(* POU FB_BACnet_MultiStateOutput_EX, ST *)
FUNCTION_BLOCK FB_BACnet_MultiStateOutput_EX
VAR_INPUT
	bEnablePV			: BOOL; (* enable present value with priority x in priority array, FALSE = priority x disable *)
	bNullPV				: BOOL; (* clear priority entry *)
	nPV					: UDINT; (* number for priority x, when input bEnablePV is TRUE *)
END_VAR
VAR_IN_OUT
	Device				: FB_BACnet_Device;
END_VAR
VAR_OUTPUT
	bReady				: BOOL;
	nPresentValue		: UDINT;
	bOverridden			: BOOL;
	bOutOfService		: BOOL;
	bFault				: BOOL;
	bInAlarm			: BOOL;
	bNoOutput			: BOOL;
	bOpenLoop			: BOOL;
	bShortedLoop		: BOOL;
	bOtherFault			: BOOL;
	eEventState			: E_BACNETEVENTSTATE;
	bAckedTrans_ToOffNormal : BOOL;
	bAckedTrans_ToFault		: BOOL;
	bAckedTrans_ToNormal	: BOOL;
	nActivePrio			: UINT;
	nNbrOfStates		: UDINT;
	tObjectID			: T_BACnet_ObjectIdentifier := 16#FFFFFFFF;
	bError				: BOOL;
	nErrorId			: UINT;
END_VAR
VAR
	_PresentValue AT%I*: UDINT; 			(* ~(BACnet_PresentValue 		:		: )
								   				(BACnet_ObjectType			: MO	: )	*)
    _PresentValue_Priority12 AT%Q*: UDINT;	(* ~(BACnet_PresentValue_Priority12		:		: )	*)
	_ActivePriority AT%I*: UDINT; 			(* ~(BACnet_ActivePriority 		:		: )	*)
	_NumberOfStates AT%I*: UDINT;			(* ~(BACnet_NumberOfStates		:		: )	*)
	_ObjectId AT%I*: DWORD;					(* ~(BACnet_ObjectIdentifier	:		: LINK) *)
	_StatusFlags AT%I*: WORD; 				(* ~(BACnet_StatusFlags			:		: )	*)
	_EventState AT%I*: WORD;				(* ~(BACnet_EventState			:		: )	*)
	_Reliability AT%I*: WORD; 				(* ~(BACnet_Reliability			:		: )	*)
	_AckedTransitions AT%I*:WORD;			(* ~(BACnet_AckedTransitions	:		: ) *)
	_AckedTransBits : ST_BACnet_EventTransitionBits;
	_nUpdateCount : UDINT := 0;
	_StatusFlagsBits : ST_BACnet_StatusFlags;
END_VAR
(* update server device *)
IF (Device._nUpdateCount = _nUpdateCount) THEN
	Device();
END_IF
(* remind current number of update counter *)
_nUpdateCount := Device._nUpdateCount;

IF Device.bFirstCycle THEN
	(* first call of the server device since reboot/reset *)
	bReady := FALSE;
	_PresentValue_Priority12 := 16#FFFFFFFF;

ELSIF (F_BACnet_GetObjType(_ObjectId) <> BACnetObjectType_MultiStateOutput) THEN
	(* wrong mapping / invalid object ID *)
	IF _ObjectId = 0 THEN
		nErrorId := BACnet_ERR_WRONG_MAPPING;
	ELSE
		nErrorId := BACnet_ERR_INVALID_OBJECTID;
	END_IF
	bReady := FALSE;

ELSIF (_StatusFlags < 4) THEN
	(* wrong mapping *)
	nErrorId := BACnet_ERR_WRONG_MAPPING;
	bReady := FALSE;

ELSIF Device.bOperational THEN
	(* ready state *)
	bReady := TRUE;
	nErrorId := BACnet_ERR_NO_ERROR;

	(* write into priority array *)
	_PresentValue_Priority12 := F_BACnet_MultiStatePV(bEnablePV, bNullPV, nPV);

	(* present value *)
	nPresentValue := _PresentValue;

	(* build bit states *)
	_StatusFlagsBits := F_BACnet_StatusFlags(_StatusFlags);
	_AckedTransBits		:= F_BACnet_EventTransitionFlags(_AckedTransitions);

	(* copy states to output *)
	bOverridden := _StatusFlagsBits.overridden;
	bOutOfService := _StatusFlagsBits.out_of_service;
	bFault := _StatusFlagsBits.fault;
	bInAlarm := _StatusFlagsBits.in_alarm;
	bNoOutput := (_Reliability = BACnetReliability_no_output);
	bOpenLoop := (_Reliability = BACnetReliability_open_loop);
	bShortedLoop := (_Reliability = BACnetReliability_shorted_loop);
	bOtherFault := (_Reliability = BACnetReliability_unreliable_other);
	bAckedTrans_ToOffNormal := _AckedTransBits.to_offnormal;
	bAckedTrans_ToFault := _AckedTransBits.to_fault;
	bAckedTrans_ToNormal := _AckedTransBits.to_normal;
	tObjectID := _ObjectId;

	(* convert enumeration *)
	eEventState := _EventState;

	(* copy active priority *)
	nActivePrio := UDINT_TO_UINT(_ActivePriority);

	(* number of states *)
	nNbrOfStates := _NumberOfStates;

ELSE
	(* server device not ready, reset local ready also *)
	bReady := FALSE;
	nErrorId := BACnet_ERR_OPERATIONAL;
END_IF
(* set error flag *)
bError := (nErrorId <> BACnet_ERR_NO_ERROR);
END_FUNCTION_BLOCK

(* POU FB_BACnet_MultiStateOutput_RAW, ST *)
FUNCTION_BLOCK FB_BACnet_MultiStateOutput_RAW
VAR_INPUT
	bEnablePV			: BOOL; (* enable present value with priority x in priority array, FALSE = priority x disable *)
	bNullPV				: BOOL; (* clear priority entry *)
	nPV					: UDINT; (* number for priority x, when input bEnablePV is TRUE *)
	nFeedback			AT%Q*: DWORD; (* ~(BACnet_FeedbackValue : : ) *)
	bNoOutput			: BOOL;
	bOpenLoop			: BOOL;
	bShortedLoop		: BOOL;
	bCommFailure		: BOOL;
	bOtherFault			: BOOL;
END_VAR
VAR_IN_OUT
	Device				: FB_BACnet_Device;
END_VAR
VAR_OUTPUT
	bReady				: BOOL;
	nPresentValue		: UDINT;
	bOverridden			: BOOL;
	bOutOfService		: BOOL;
	bFault				: BOOL;
	bInAlarm			: BOOL;
	bAckedTrans_ToOffNormal : BOOL;
	bAckedTrans_ToFault		: BOOL;
	bAckedTrans_ToNormal	: BOOL;
	nNbrOfStates		: UDINT;
	bError				: BOOL;
	nErrorId			: UINT;
	nRawOut				AT%I*: DWORD;		(* ~(BACnet_PresentValue		:		: ) *)
END_VAR
VAR
    _PresentValue_Priority12 AT%Q*: UDINT;	(* ~(BACnet_PresentValue_Priority12:	: )
								   				(BACnet_ObjectType			: MO	: )	*)
	_Reliability AT%Q*: WORD := BACnetReliability_no_fault_detected;(* ~(BACnet_Reliability 	:		: )	*)
	_NumberOfStates AT%I*: UDINT;			(* ~(BACnet_NumberOfStates		:		: )	*)
	_ObjectId AT%I*: DWORD;					(* ~(BACnet_ObjectIdentifier	:		: LINK) *)
	_StatusFlags AT%I*: WORD; 				(* ~(BACnet_StatusFlags			:		: )	*)
	_AckedTransitions AT%I*:WORD;			(* ~(BACnet_AckedTransitions	:		: ) *)
	_AckedTransBits : ST_BACnet_EventTransitionBits;
	_nUpdateCount : UDINT := 0;
	_StatusFlagsBits : ST_BACnet_StatusFlags;
END_VAR
(* update server device *)
IF (Device._nUpdateCount = _nUpdateCount) THEN
	Device();
END_IF
(* remind current number of update counter *)
_nUpdateCount := Device._nUpdateCount;

(* handle raw error *)
IF bNoOutput THEN
	_Reliability := BACnetReliability_no_output;
ELSIF bOpenLoop THEN
	_Reliability := BACnetReliability_open_loop;
ELSIF bShortedLoop THEN
	_Reliability := BACnetReliability_shorted_loop;
ELSIF bCommFailure THEN
	_Reliability := BACnetReliability_communication_failure;
ELSIF bOtherFault THEN
	_Reliability := BACnetReliability_unreliable_other;
ELSE
	_Reliability := BACnetReliability_no_fault_detected;
END_IF

(* check object type *)
IF Device.bFirstCycle THEN
	(* first call of the server device since reboot/reset *)
	bReady := FALSE;
	_PresentValue_Priority12 := 16#FFFFFFFF;

ELSIF (F_BACnet_GetObjType(_ObjectId) <> BACnetObjectType_MultiStateOutput) THEN
	(* wrong mapping / invalid object ID *)
	IF _ObjectId = 0 THEN
		nErrorId := BACnet_ERR_WRONG_MAPPING;
	ELSE
		nErrorId := BACnet_ERR_INVALID_OBJECTID;
	END_IF
	bReady := FALSE;

ELSIF (_StatusFlags < 4) THEN
	(* wrong mapping *)
	nErrorId := BACnet_ERR_WRONG_MAPPING;
	bReady := FALSE;

ELSIF Device.bOperational THEN
	(* ready state *)
	bReady := TRUE;
	nErrorId := BACnet_ERR_NO_ERROR;

	(* write into priority array *)
	_PresentValue_Priority12 := F_BACnet_MultiStatePV(bEnablePV, bNullPV, nPV);

	(* present value *)
	nPresentValue := nRawOut;

	(* build bit states *)
	_StatusFlagsBits := F_BACnet_StatusFlags(_StatusFlags);
	_AckedTransBits		:= F_BACnet_EventTransitionFlags(_AckedTransitions);

	(* copy states to output *)
	bOverridden := _StatusFlagsBits.overridden;
	bOutOfService := _StatusFlagsBits.out_of_service;
	bFault := _StatusFlagsBits.fault;
	bInAlarm := _StatusFlagsBits.in_alarm;
	bAckedTrans_ToOffNormal := _AckedTransBits.to_offnormal;
	bAckedTrans_ToFault := _AckedTransBits.to_fault;
	bAckedTrans_ToNormal := _AckedTransBits.to_normal;

	(* number of states *)
	nNbrOfStates := _NumberOfStates;

ELSE
	(* server device not ready, reset local ready also *)
	bReady := FALSE;
	nErrorId := BACnet_ERR_OPERATIONAL;
END_IF
(* set error flag *)
bError := (nErrorId <> BACnet_ERR_NO_ERROR);
END_FUNCTION_BLOCK

(* POU FB_BACnet_MultiStateValue, ST *)
FUNCTION_BLOCK FB_BACnet_MultiStateValue
VAR_INPUT
	bEnablePV		: BOOL; (* enable present value with priority x in priority array, FALSE = priority x disable *)
	bNullPV			: BOOL; (* clear priority entry *)
	nPV				: UDINT; (* number for priority x, when input bEnablePV is TRUE *)
END_VAR
VAR_IN_OUT
	Device	: FB_BACnet_Device;
END_VAR
VAR_OUTPUT
	bReady			: BOOL;
	nPresentValue	: UDINT;
	bOverridden		: BOOL;
	bOutOfService	: BOOL;
	bFault			: BOOL;
	bInAlarm		: BOOL;
	nNbrOfStates	: UDINT;
	bError			: BOOL;
	nErrorId		: UINT;
END_VAR
VAR
	_PresentValue AT%I*: UDINT; 			(* ~(BACnet_PresentValue 		:		: )
								   				(BACnet_ObjectType 			: MV	: )	*)
	_NumberOfStates AT%I*: UDINT;			(* ~(BACnet_NumberOfStates		:		: )	*)
	_StatusFlags AT%I*: WORD; 				(* ~(BACnet_StatusFlags 		:		: )	*)
    _PresentValue_Priority12 AT%Q*: UDINT;	(* ~(BACnet_PresentValue_Priority12:	: )	*)
	_nUpdateCount : UDINT := 0;
	_StatusFlagsBits : ST_BACnet_StatusFlags;
END_VAR
(* update server device *)
IF (Device._nUpdateCount = _nUpdateCount) THEN
	Device();
END_IF
(* remind current number of update counter *)
_nUpdateCount := Device._nUpdateCount;

IF Device.bFirstCycle THEN
	(* first call of the server device since reboot/reset *)
	bReady := FALSE;
	_PresentValue_Priority12 := 16#FFFFFFFF;

ELSIF (_StatusFlags < 4) THEN
	(* wrong mapping *)
	nErrorId := BACnet_ERR_WRONG_MAPPING;
	bReady := FALSE;

ELSIF Device.bOperational THEN
	(* ready state *)
	bReady := TRUE;
	nErrorId := BACnet_ERR_NO_ERROR;

	(* write into priority array *)
	_PresentValue_Priority12 := F_BACnet_MultiStatePV(bEnablePV, bNullPV, nPV);

	(* present value *)
	nPresentValue := _PresentValue;

	(* build bit states *)
	_StatusFlagsBits := F_BACnet_StatusFlags(_StatusFlags);

	(* copy states to output *)
	bOverridden := _StatusFlagsBits.overridden;
	bOutOfService := _StatusFlagsBits.out_of_service;
	bFault := _StatusFlagsBits.fault;
	bInAlarm := _StatusFlagsBits.in_alarm;

	(* number of states *)
	nNbrOfStates := _NumberOfStates;

ELSE
	(* server device not ready, reset local ready also *)
	bReady := FALSE;
	nErrorId := BACnet_ERR_OPERATIONAL;
END_IF
(* set error flag *)
bError := (nErrorId <> BACnet_ERR_NO_ERROR);
END_FUNCTION_BLOCK

(* POU FB_BACnet_MultiStateValue_ADS, ST *)
FUNCTION_BLOCK FB_BACnet_MultiStateValue_ADS
VAR_INPUT
	bEnablePV			: BOOL; (* enable PV write commands *)
	bNullPV				: BOOL; (* clear priority entry *)
	nPV					: UDINT; (* number for priority x, when input bEnablePV is TRUE and bNullPV is FALSE *)
	bManual				: BOOL; (* FALSE --> TRUE: write present_value immediately, FALSE: only write present_value on-change, TRUE: write present_value on-change and when device turns operational *)
	ePriority			: E_BACNETPRIORITY := BACNETPRIORITY_12;
END_VAR
VAR_IN_OUT
	Device				: FB_BACnet_Device;
END_VAR
VAR_OUTPUT
	bReady				: BOOL;
	bPvDone				: BOOL; (* present_value written over ADS *)
	nPresentValue		: UDINT;
	bOverridden			: BOOL;
	bOutOfService		: BOOL;
	bFault				: BOOL;
	bInAlarm			: BOOL;
	nNbrOfStates		: UDINT;
	tObjectID			: T_BACnet_ObjectIdentifier := 16#FFFFFFFF;
	bError				: BOOL;
	nErrorId			: UINT;
	nAdsErrorId			: UDINT;
END_VAR
VAR
	_StatusFlags AT%I*: WORD; 				(* ~(BACnet_StatusFlags 	:		: )	*)
	_PresentValue AT%I*: UDINT; 			(* ~(BACnet_PresentValue 	:		: )
								   				(BACnet_ObjectType 		: MV	: )	*)
	_NumberOfStates AT%I*: UDINT;			(* ~(BACnet_NumberOfStates	:		: )	*)
	_ObjectId AT%I*: DWORD;					(* ~(BACnet_ObjectIdentifier:		: LINK) *)
	_StatusFlagsBits : ST_BACnet_StatusFlags;
    _PresentValue_Ads : UDINT;
	_nUpdateCount : UDINT := 0;
	_WriteProp : FB_BACnet_WriteProp;
	_rtrigManual : R_TRIG;
	_bNullPvOld : BOOL;
	_nObjType : E_BACNETOBJECTTYPE;
END_VAR
(* update server device *)
IF (Device._nUpdateCount = _nUpdateCount) THEN
	Device();
END_IF
(* remind current number of update counter *)
_nUpdateCount := Device._nUpdateCount;

(* trigger on manual flag *)
_rtrigManual(CLK:= bManual, Q=> );

(* decode object type *)
_nObjType := F_BACnet_GetObjType(_ObjectId);

IF Device.bFirstCycle THEN
	(* first call of the server device since reboot/reset *)
	bReady := FALSE;
	bPvDone := FALSE;

ELSIF _nObjType <> BACnetObjectType_MultiStateValue THEN
	(* wrong mapped object type *)
	nErrorId := BACnet_ERR_INVALID_OBJECTTYPE;
	bReady := FALSE;
	bPvDone := FALSE;

ELSIF (_StatusFlags < 4) THEN
	(* wrong mapping *)
	nErrorId := BACnet_ERR_WRONG_MAPPING;
	bReady := FALSE;
	bPvDone := FALSE;

ELSIF Device.bOperational THEN

	IF Device.stAdsConn.bValid THEN
		(* write present_value on manual trigger, on-change and on operational recover *)
		IF		bEnablePV
			AND	(		_rtrigManual.Q
					OR	(nPV <> _PresentValue_Ads)
					OR	((NOT bReady) AND bManual)
					OR	(bNullPV <> _bNullPvOld)
				)
		THEN
			_WriteProp.bExecute := TRUE;
			bPvDone := FALSE;
			(* write depending on enable state *)
			IF bNullPV THEN
				_PresentValue_Ads := 0;
			ELSE
				_PresentValue_Ads := nPV;
			END_IF
			_bNullPvOld := bNullPV;
		END_IF

		(* ready state *)
		IF (nAdsErrorId = 0) THEN
			bReady := TRUE;
			nErrorId := BACnet_ERR_NO_ERROR;
		END_IF

	ELSE
		(* invalid ADS connection *)
		bReady := FALSE;
		nErrorId := BACnet_ERR_INVALID_ADS_CONN;
		bPvDone := FALSE;
	END_IF

	(* present value *)
	nPresentValue := _PresentValue;

	(* build bit states *)
	_StatusFlagsBits := F_BACnet_StatusFlags(_StatusFlags);

	(* copy states to output *)
	bOverridden := _StatusFlagsBits.overridden;
	bOutOfService := _StatusFlagsBits.out_of_service;
	bFault := _StatusFlagsBits.fault;
	bInAlarm := _StatusFlagsBits.in_alarm;
	tObjectID := _ObjectId;

	(* number of states *)
	nNbrOfStates := _NumberOfStates;

ELSE
	(* server device not ready, reset local ready also *)
	bReady := FALSE;
	nErrorId := BACnet_ERR_OPERATIONAL;
	bPvDone := FALSE;
END_IF

(* call write property command *)
_WriteProp(
	BACnetDevicePort	:= Device.stAdsConn.nAmsPort,
	bExecute			:= ,
	sNetId				:= Device.stAdsConn.sAmsNetId,
	ObjectType			:= _nObjType,
	PropertyID			:= BACnetPropertyIdentifier_PresentValue,
	Priority			:= ePriority,
	DataType			:= BACnetDataType_UnsignedInteger,
	ObjectInstance		:= F_BACnet_GetObjInstance(_ObjectId),
	ptrValue			:= ADR(_PresentValue_Ads),
	nLenValue			:= SIZEOF(_PresentValue_Ads),
	bDone				=> ,
	bBusy				=> ,
	bError				=> ,
	nErrID				=> );

(* set done flag *)
IF _WriteProp.bExecute AND (NOT _WriteProp.bBusy) THEN
	(* check if command was finished with error *)
	IF _WriteProp.bError THEN
		bPvDone		:= FALSE;
		bReady		:= FALSE;
		nErrorId	:= BACnet_ERR_ADS_Write;
	ELSE
		(* successful written *)
		bPvDone		:= TRUE;
	END_IF
	nAdsErrorId := _WriteProp.nErrID;
	(* reset execution bit *)
	_WriteProp(bExecute := FALSE);
END_IF

(* set error flag *)
bError := (nErrorId <> BACnet_ERR_NO_ERROR) OR (nAdsErrorId <> 0);
END_FUNCTION_BLOCK

(* POU FB_BACnet_MultiStateValue_EX, ST *)
FUNCTION_BLOCK FB_BACnet_MultiStateValue_EX
VAR_INPUT
	bEnablePV			: BOOL; (* enable present value with priority x in priority array, FALSE = priority x disable *)
	bNullPV				: BOOL; (* clear priority entry *)
	nPV					: UDINT; (* number for priority x, when input bEnablePV is TRUE *)
END_VAR
VAR_IN_OUT
	Device				: FB_BACnet_Device;
END_VAR
VAR_OUTPUT
	bReady				: BOOL;
	nPresentValue		: UDINT;
	bOverridden			: BOOL;
	bOutOfService		: BOOL;
	bFault				: BOOL;
	bInAlarm			: BOOL;
	bMultiStateFault	: BOOL;
	bOtherFault			: BOOL;
	eEventState			: E_BACNETEVENTSTATE;
	bAckedTrans_ToOffNormal : BOOL;
	bAckedTrans_ToFault		: BOOL;
	bAckedTrans_ToNormal	: BOOL;
	nActivePrio			: UINT;
	nNbrOfStates		: UDINT;
	tObjectID			: T_BACnet_ObjectIdentifier := 16#FFFFFFFF;
	bError				: BOOL;
	nErrorId			: UINT;
END_VAR
VAR
	_PresentValue AT%I*: UDINT; 			(* ~(BACnet_PresentValue 	:		: )
								   				(BACnet_ObjectType 		: MV	: )	*)
    _PresentValue_Priority12 AT%Q*: UDINT;	(* ~(BACnet_PresentValue_Priority12	:		: )	*)
	_ActivePriority AT%I*: UDINT; 			(* ~(BACnet_ActivePriority 	:		: )	*)
	_NumberOfStates AT%I*: UDINT;			(* ~(BACnet_NumberOfStates	:		: )	*)
	_ObjectId AT%I*: DWORD;					(* ~(BACnet_ObjectIdentifier:		: LINK) *)
	_StatusFlags AT%I*: WORD; 				(* ~(BACnet_StatusFlags 	:		: )	*)
	_EventState AT%I*: WORD;				(* ~(BACnet_EventState 		:		: )	*)
	_Reliability AT%I*: WORD;				(* ~(BACnet_Reliability 	:		: )	*)
	_AckedTransitions AT%I*:WORD;			(* ~(BACnet_AckedTransitions:		: ) *)
	_AckedTransBits : ST_BACnet_EventTransitionBits;
	_StatusFlagsBits : ST_BACnet_StatusFlags;
	_nUpdateCount : UDINT := 0;
END_VAR
(* update server device *)
IF (Device._nUpdateCount = _nUpdateCount) THEN
	Device();
END_IF
(* remind current number of update counter *)
_nUpdateCount := Device._nUpdateCount;

IF Device.bFirstCycle THEN
	(* first call of the server device since reboot/reset *)
	bReady := FALSE;
	_PresentValue_Priority12 := 16#FFFFFFFF;

ELSIF (F_BACnet_GetObjType(_ObjectId) <> BACnetObjectType_MultiStateValue) THEN
	(* wrong mapping / invalid object ID *)
	IF _ObjectId = 0 THEN
		nErrorId := BACnet_ERR_WRONG_MAPPING;
	ELSE
		nErrorId := BACnet_ERR_INVALID_OBJECTID;
	END_IF
	bReady := FALSE;

ELSIF (_StatusFlags < 4) THEN
	(* wrong mapping *)
	nErrorId := BACnet_ERR_WRONG_MAPPING;
	bReady := FALSE;

ELSIF Device.bOperational THEN
	(* ready state *)
	bReady := TRUE;
	nErrorId := BACnet_ERR_NO_ERROR;

	(* write into priority array *)
	_PresentValue_Priority12 := F_BACnet_MultiStatePV(bEnablePV, bNullPV, nPV);

	(* present value *)
	nPresentValue := _PresentValue;

	(* build bit states *)
	_StatusFlagsBits := F_BACnet_StatusFlags(_StatusFlags);
	_AckedTransBits		:= F_BACnet_EventTransitionFlags(_AckedTransitions);

	(* copy states to output *)
	bOverridden := _StatusFlagsBits.overridden;
	bOutOfService := _StatusFlagsBits.out_of_service;
	bFault := _StatusFlagsBits.fault;
	bInAlarm := _StatusFlagsBits.in_alarm;
	bMultiStateFault := (_Reliability = BACnetReliability_multi_state_fault);
	bOtherFault := (_Reliability = BACnetReliability_unreliable_other);
	bAckedTrans_ToOffNormal := _AckedTransBits.to_offnormal;
	bAckedTrans_ToFault := _AckedTransBits.to_fault;
	bAckedTrans_ToNormal := _AckedTransBits.to_normal;
	tObjectID := _ObjectId;

	(* convert enumeration *)
	eEventState := _EventState;

	(* copy active priority *)
	nActivePrio := UDINT_TO_UINT(_ActivePriority);

	(* number of states *)
	nNbrOfStates := _NumberOfStates;

ELSE
	(* server device not ready, reset local ready also *)
	bReady := FALSE;
	nErrorId := BACnet_ERR_OPERATIONAL;
END_IF
(* set error flag *)
bError := (nErrorId <> BACnet_ERR_NO_ERROR);
END_FUNCTION_BLOCK

(* POU FB_BACnet_NotificationClass, ST *)
FUNCTION_BLOCK FB_BACnet_NotificationClass
VAR_IN_OUT
	Device	: FB_BACnet_Device;
END_VAR
VAR_OUTPUT
	bReady			: BOOL;
	bError			: BOOL;
	nErrorId		: UINT;
END_VAR
VAR
	_ObjectId AT%I* : DWORD;					(* ~(BACnet_ObjectIdentifier:		: LINK)
													(BACnet_ObjectType		:	NC	: ) *)
	_nUpdateCount	: UDINT := 0;
END_VAR
(* update server device *)
IF (Device._nUpdateCount = _nUpdateCount) THEN
	Device();
END_IF
(* remind current number of update counter *)
_nUpdateCount := Device._nUpdateCount;

IF Device.bOperational THEN
	(* ready state *)
	bReady := TRUE;
	nErrorId := BACnet_ERR_NO_ERROR;
ELSE
	(* server device not ready, reset local ready also *)
	bReady := FALSE;
	nErrorId := BACnet_ERR_OPERATIONAL;
END_IF
(* set error flag *)
bError := (nErrorId <> BACnet_ERR_NO_ERROR);
END_FUNCTION_BLOCK

(* POU FB_BACnet_NotificationClass_EX, ST *)
FUNCTION_BLOCK FB_BACnet_NotificationClass_EX
VAR_IN_OUT
	Device				: FB_BACnet_Device;
END_VAR
VAR_OUTPUT
	bReady				: BOOL;
	tObjectID			: T_BACnet_ObjectIdentifier := 16#FFFFFFFF;
	bError				: BOOL;
	nErrorId			: UINT;
END_VAR
VAR
	_ObjectId AT%I* : DWORD;					(* ~(BACnet_ObjectIdentifier:		: LINK)
													(BACnet_ObjectType		:	NC	: ) *)
	_nUpdateCount	: UDINT := 0;
END_VAR
(* update server device *)
IF (Device._nUpdateCount = _nUpdateCount) THEN
	Device();
END_IF
(* remind current number of update counter *)
_nUpdateCount := Device._nUpdateCount;

IF (F_BACnet_GetObjType(_ObjectId) <> BACnetObjectType_NotificationClass) THEN
	(* wrong mapping / invalid object ID *)
	IF _ObjectId = 0 THEN
		nErrorId := BACnet_ERR_WRONG_MAPPING;
	ELSE
		nErrorId := BACnet_ERR_INVALID_OBJECTID;
	END_IF
	bReady := FALSE;
	tObjectID := 16#FFFFFFFF;

ELSIF Device.bOperational THEN
	(* ready state *)
	bReady := TRUE;
	nErrorId := BACnet_ERR_NO_ERROR;
	tObjectID := _ObjectId;

ELSE
	(* server device not ready, reset local ready also *)
	bReady := FALSE;
	nErrorId := BACnet_ERR_OPERATIONAL;
END_IF
(* set error flag *)
bError := (nErrorId <> BACnet_ERR_NO_ERROR);
END_FUNCTION_BLOCK

(* POU FB_BACnet_NotificationSink, ST *)
FUNCTION_BLOCK FB_BACnet_NotificationSink
VAR_INPUT
	bReload			: BOOL;
	nAmsPort		: T_AmsPort := 0;
END_VAR
VAR_OUTPUT
	bReady			: BOOL;
	stBACnetAds		: ST_BACnet_AdsConnection;
END_VAR
VAR
	_rtrigReload	: R_TRIG;
	_nUpdateCountAdp: UDINT := 0;
	_BACnetAdapter	: POINTER TO FB_BACnet_Adapter;
END_VAR
(* check pointer to bacnet adapter instance *)
IF pBACnet_Adapter > 0 THEN
	_BACnetAdapter := pBACnet_Adapter;
ELSE
	_BACnetAdapter := ADR(fbBACnet_Adapter);
END_IF

(* update adapter *)
IF _BACnetAdapter^._nUpdateCount = _nUpdateCountAdp THEN
	_BACnetAdapter^();
END_IF
(* remind current number of update counter *)
_nUpdateCountAdp := _BACnetAdapter^._nUpdateCount;

(* set ads info *)
stBACnetAds.nAmsPort := nAmsPort;
stBACnetAds.bNSink := TRUE;
stBACnetAds.bServer := FALSE;
stBACnetAds.bClient := FALSE;
stBACnetAds.nDeviceId := 16#FFFFFFFF;
stBACnetAds.sAmsNetId := _BACnetAdapter^.sAmsNetId;
bReady := stBACnetAds.bValid;
stBACnetAds.bValid :=	(nAmsPort >= 1000) AND (nAmsPort < 16#FFFF)
					AND	(_BACnetAdapter^.eAdapterStatus > BACnetAdapterStatus_Init);

(* set reload counter *)
_rtrigReload(CLK:= bReload, Q=> );
IF stBACnetAds.bValid AND (_rtrigReload.Q OR (NOT bReady)) THEN
	stBACnetAds.nReload := stBACnetAds.nReload + 1;
END_IF

(* set states *)
bReady := stBACnetAds.bValid;
END_FUNCTION_BLOCK

(* POU FB_BACnet_NotificationSinkDelEntry, ST *)
FUNCTION_BLOCK FB_BACnet_NotificationSinkDelEntry
VAR_INPUT
	bExecute	: BOOL;
	nIndex		: UDINT;
	sNetId		: T_AmsNetId;
	nPort		: T_AmsPort;
	tTimeout	: TIME := BACnet_ADSTimeOut;
END_VAR
VAR_OUTPUT
	bBusy		: BOOL;
	bEmpty		: BOOL;
	bError		: BOOL;
	nErrorId	: UDINT;
END_VAR
VAR
	_AdsReadClient	: ADSREAD;
END_VAR
	_AdsReadClient(
		NETID	:= sNetId,
		PORT	:= nPort,
		IDXGRP	:= 16#5,
		IDXOFFS	:= nIndex,
		LEN		:= 0,
		DESTADDR:= 0,
		READ	:= bExecute,
		TMOUT	:= tTimeout,
		BUSY	=> bBusy,
		ERR		=> bError,
		ERRID	=> nErrorId);

	bEmpty := ((UDINT_TO_DWORD(_AdsReadClient.ERRID) AND 16#FFF) = 16#703);
END_FUNCTION_BLOCK

(* POU FB_BACnet_NSinkAcknEvent, ST *)
FUNCTION_BLOCK FB_BACnet_NSinkAcknEvent
VAR_INPUT
	bAcknowledge	: BOOL;
	stAcknEvent		: ST_BACnet_NSinkEvent;
	sMessage		: T_MaxString;
END_VAR
VAR_IN_OUT
	stAdsConn		: ST_BACnet_AdsConnection;
END_VAR
VAR_OUTPUT
	bDone			: BOOL;
	bBusy			: BOOL;
	bError			: BOOL;
	nErrorId		: UINT;
END_VAR
VAR
	_fbAdsWrite		: FW_AdsWrite;
	_i				: INT;
	_rtrigGetSet	: R_TRIG;
	_stNSinkRawData	: ST_BACnet_NotificationSinkEventEntry;
	_stringEncode	: FB_BACnet_StringExtEncode;
	_pChrStringExt	: POINTER TO ST_BACnet_CharacterStringExt;
END_VAR
(*

#define BACNET_STRING_MAXLENGTH    256

typedef struct _EventNotificationRequest
{
      ULONG validFields;
      ULONG processIdentifier;
      BACnetObjectIdentifier initiatingDeviceIdentifier;
      BACnetObjectIdentifier eventObjectIdentifier;
      BACnetTimeStamp timeStamp;
      ULONG notificationClass;
      ULONG priority;
      BACnetEventType eventType;
      CHAR messageText[BACNET_STRING_MAXLENGTH];
      BACnetNotifyType notifyType;
      BOOL ackRequired;
      BACnetEventState fromState;
      BACnetEventState toState;
      PBACnetNotificationParameters pEventValues;
}EventNotificationRequest, *PEventNotificationRequest;

*)

(* ADS write *)
_fbAdsWrite(
	sNetId		:= stAdsConn.sAmsNetId,
	nPort		:= stAdsConn.nAmsPort,
	nIdxGrp		:= BACnet_ADSIGRP_NTFSINK_W_EVENTNTF_ACK_BY_PARAMETER,
	nIdxOffs	:= 0,
	cbWriteLen	:= SIZEOF(_stNSinkRawData) - SIZEOF(_stNSinkRawData._fillBytes00),
	pWriteBuff	:= ADR(_stNSinkRawData.validFields),
	bExecute	:= ,
	tTimeout	:= BACnet_ADSTimeOut,
	bBusy		=> ,
	bError		=> ,
	nErrId		=> );

(* trigger start event *)
_rtrigGetSet(CLK:= bAcknowledge, Q=> );

(* state machine *)
CASE _i OF

	0: (* Idle *)
		IF _rtrigGetSet.Q THEN
			IF (NOT stAdsConn.bValid) THEN
				(* ADS connection not valid *)
				nErrorId := BACnet_ERR_INVALID_ADS_CONN;
			ELSIF (NOT stAdsConn.bNSink) THEN
				(* not a notification sink *)
				nErrorId := BACnet_ERR_ADS_NoNotificationSink;
			ELSE
				nErrorId := BACnet_ERR_NO_ERROR;
				_i := 1;
				(* prepare raw data *)
				MEMSET(destAddr:=ADR(_stNSinkRawData), fillByte:=0, n:=SIZEOF(_stNSinkRawData));
				(* encode message text to UTF-8 *)
				_stringEncode(
					pString			:= ADR(sMessage),
					nSize			:= LEN(sMessage),
					pResultExtStr	:= ADR(_stNSinkRawData.messageText),
					cbResult		:= SIZEOF(_stNSinkRawData.messageText),
					bValid			=> ,
					bOverflow		=> ,
					nLength			=> );
				(* fill flags and other information *)
				_stNSinkRawData.ackRequired := FALSE;
				_stNSinkRawData.eventObjectIdentifier := stAcknEvent.tObjectID;
				_stNSinkRawData.eventType := stAcknEvent.eEventType;
				_stNSinkRawData.fromState := stAcknEvent.eFromState;
				_stNSinkRawData.toState := stAcknEvent.eToState;
				_stNSinkRawData.initiatingDeviceIdentifier := stAcknEvent.nDeviceID;
				_stNSinkRawData.notificationClass := stAcknEvent.nNC;
				_stNSinkRawData.notifyType := BACnetNotifyType_ack_notification;
				_stNSinkRawData.priority := stAcknEvent.nPriotity;
				_stNSinkRawData.processIdentifier := stAcknEvent.nProcessID;
				_stNSinkRawData.timeStamp.stDateTime := stAcknEvent.stDateTime;
				_stNSinkRawData.timeStamp.eType := BACnetTimeStampChoice_dateTime;
			END_IF
			(* reset done flag *)
			bDone := FALSE;
		END_IF
		IF (NOT bAcknowledge) THEN
			nErrorId := BACnet_ERR_NO_ERROR;
			bDone := FALSE;
		END_IF

	(* WRITE *)
	1: (* write data over ADS *)
		IF _fbAdsWrite.bExecute THEN
			IF _fbAdsWrite.bError THEN
				_i := 100;
				nErrorId := BACnet_ERR_ADS_Write;
				_fbAdsWrite.bExecute := FALSE;
			ELSIF (NOT _fbAdsWrite.bBusy) THEN
				(* DONE *)
				_fbAdsWrite.bExecute := FALSE;
				_i := 100;
			END_IF
		ELSE
			_fbAdsWrite.bExecute := TRUE;
		END_IF

	100: (* Done *)
		bDone := (nErrorId = BACnet_ERR_NO_ERROR);
		_i := 0;

END_CASE

(* set error flag *)
bError 	:= nErrorId > BACnet_ERR_NO_ERROR;
bBusy 	:= _i > 0;
END_FUNCTION_BLOCK

(* POU FB_BACnet_StringExtEncode, ST *)
FUNCTION_BLOCK FB_BACnet_StringExtEncode (* convert Windows-1252 to ANSI/UTF-8 BACnet Character String *)
VAR_INPUT
	pString			: POINTER TO T_MaxString; (* pointer to Windows-1252 encoded PLC text *)
	nSize			: INT; (* string length or data size of pText field *)
	pResultExtStr	: POINTER TO ST_BACnet_CharacterStringExt;
	cbResult		: UDINT; (* byte size of result data field *)
END_VAR
VAR_OUTPUT
	bValid			: BOOL;
	bOverflow		: BOOL; (* String length overflow (source string too long) *)
	nLength			: UDINT; (* out string data length in byte *)
END_VAR
(* preset valid to FALSE *)
bOverflow := FALSE;
bValid := TRUE;
(* check pointer *)
IF (pString = 0) OR (pResultExtStr = 0) THEN
	nLength := 0;
	bValid := FALSE;
	RETURN;
END_IF

(* clear string *)
MEMSET(destAddr:=pResultExtStr, fillByte:=0, n:=cbResult);
(* check input size *)
IF (nSize <= 0) THEN
	nLength := 0;

(* convert *)
ELSE
	IF (_F_BACnet_EncodeUTF8(
		pString		:= pString,
		cbString	:= nSize,
		pResult		:= pResultExtStr,
		cbResult	:= cbResult,
		nResultLen	:= nLength) > cbResult)
	THEN
		bOverflow	:= TRUE;
		bValid		:= FALSE;
	END_IF
END_IF
END_FUNCTION_BLOCK

(* POU FB_BACnet_NSinkReadEvent, ST *)
FUNCTION_BLOCK FB_BACnet_NSinkReadEvent
VAR_INPUT
	nIndex			: UDINT;
	bAutoGet		: BOOL:=TRUE; (* TRUE = get data when ADS connection or index changed *)
	bGet			: BOOL; (* FALSE --> TRUE = get data from property *)
END_VAR
VAR_IN_OUT
	stAdsConn		: ST_BACnet_AdsConnection;
END_VAR
VAR_OUTPUT
	bDone			: BOOL;
	bNoEntry		: BOOL;
	bBusy			: BOOL;
	bError			: BOOL;
	nErrorId		: UINT;
	stEvent			: ST_BACnet_NSinkEvent;
END_VAR
VAR
	_fbAdsRead		: FW_AdsRead;
	_i				: INT;
	_nOldIndex		: UDINT;
	_rtrigGetSet	: R_TRIG;
	_nAdsReloadOld	: USINT;
	_stNSinkRawData	: ST_BACnet_NotificationSinkEventEntry;
	_StringExtDecode: FB_BACnet_StringExtDecode;
END_VAR
(*

#define BACNET_STRING_MAXLENGTH    256


enum EventNotificationRequestFields
{
      notify_processIdentifier,
      notify_initiatingDeviceIdentifier,
      notify_eventObjectIdentifier,
      notify_timeStamp,
      notify_notificationClass,
      notify_priority,
      notify_eventType,
      notify_messageText,
      notify_notifyType,
      notify_ackRequired,
      notify_fromState,
      notify_toState,
      notify_eventValues,
};

typedef struct _EventNotificationRequest
{
      ULONG validFields;
      ULONG processIdentifier;
      BACnetObjectIdentifier initiatingDeviceIdentifier;
      BACnetObjectIdentifier eventObjectIdentifier;
      BACnetTimeStamp timeStamp;
      ULONG notificationClass;
      ULONG priority;
      BACnetEventType eventType;
      CHAR messageText[BACNET_STRING_MAXLENGTH];
      BACnetNotifyType notifyType;
      BOOL ackRequired;
      BACnetEventState fromState;
      BACnetEventState toState;
      PBACnetNotificationParameters pEventValues;
}EventNotificationRequest, *PEventNotificationRequest;


*)

(* ADS read *)
_fbAdsRead(
	sNetId		:= stAdsConn.sAmsNetId,
	nPort		:= stAdsConn.nAmsPort,
	nIdxGrp		:= BACnet_ADSIGRP_NTFSINK_EVENTNTF_READ,
	nIdxOffs	:= nIndex,
	cbReadLen	:= SIZEOF(_stNSinkRawData),
	pReadBuff	:= ADR(_stNSinkRawData),
	bExecute	:= ,
	tTimeout	:= BACnet_ADSTimeOut,
	bBusy		=> ,
	bError		=> ,
	nErrId		=> ,
	cbRead		=> );

(* trigger start event *)
_rtrigGetSet(CLK:= bGet, Q=> );

(* state machine *)
CASE _i OF

	0: (* Idle *)
		IF		(		(		_rtrigGetSet.Q
							OR	(_nAdsReloadOld <> stAdsConn.nReload)
							OR	(_nOldIndex <> nIndex)
						)
					AND	bAutoGet
				)
			OR	_rtrigGetSet.Q
		THEN
			IF (NOT stAdsConn.bValid) THEN
				(* ADS connection not valid *)
				nErrorId := BACnet_ERR_INVALID_ADS_CONN;
			ELSIF (NOT stAdsConn.bNSink) THEN
				(* not a notification sink *)
				nErrorId := BACnet_ERR_ADS_NoNotificationSink;
			ELSE
				nErrorId := BACnet_ERR_NO_ERROR;
				_i := 1;
				MEMSET(destAddr:=ADR(_stNSinkRawData), fillByte:=0, n:=SIZEOF(_stNSinkRawData));
				(* remind ADS reload counter and parameter *)
				_nAdsReloadOld := stAdsConn.nReload;
				_nOldIndex := nIndex;
			END_IF
			(* reset done flag *)
			bDone := FALSE;
			bNoEntry := FALSE;
		END_IF
		IF (NOT bGet) AND (NOT bAutoGet) THEN
			nErrorId := BACnet_ERR_NO_ERROR;
			bDone := FALSE;
		END_IF

	(* READ *)
	1: (* read data over ADS *)
		IF _fbAdsRead.bExecute THEN
			IF _fbAdsRead.bError THEN
				_i := 100;
				(* entry exists? *)
				bNoEntry := ((UDINT_TO_DWORD(_fbAdsRead.nErrId) AND 16#FFF) = 16#703);
				IF (NOT bNoEntry) THEN
					nErrorId := BACnet_ERR_ADS_Read;
				END_IF
				_fbAdsRead.bExecute := FALSE;
			ELSIF (NOT _fbAdsRead.bBusy) THEN
				_fbAdsRead.bExecute := FALSE;
				(* check size *)
				IF (_fbAdsRead.cbRead < 312) THEN
					(* wrong data size *)
					nErrorId := BACnet_ERR_ADS_Data;
				ELSE
					(* get the valid fields info *)
					stEvent.stValidFields.bProcessIdentifier			:= _stNSinkRawData.validFields.0;
					stEvent.stValidFields.bInitiatingDeviceIdentifier	:= _stNSinkRawData.validFields.1;
					stEvent.stValidFields.bEventObjectIdentifier		:= _stNSinkRawData.validFields.2;
					stEvent.stValidFields.bTimeStamp					:= _stNSinkRawData.validFields.3;
					stEvent.stValidFields.bNotificationClass			:= _stNSinkRawData.validFields.4;
					stEvent.stValidFields.bPriority						:= _stNSinkRawData.validFields.5;
					stEvent.stValidFields.bEventType					:= _stNSinkRawData.validFields.6;
					stEvent.stValidFields.bMessageText					:= _stNSinkRawData.validFields.7;
					stEvent.stValidFields.bNotifyType					:= _stNSinkRawData.validFields.8;
					stEvent.stValidFields.bAckRequired					:= _stNSinkRawData.validFields.9;
					stEvent.stValidFields.bFromState					:= _stNSinkRawData.validFields.10;
					stEvent.stValidFields.bToState						:= _stNSinkRawData.validFields.11;
					stEvent.stValidFields.bEventValues					:= _stNSinkRawData.validFields.12;
					(* copy data according to event valid flags *)
					IF (stEvent.stValidFields.bAckRequired) THEN
						stEvent.bAcknReq := _stNSinkRawData.ackRequired;
					END_IF
					IF (stEvent.stValidFields.bEventType) THEN
						stEvent.eEventType := _stNSinkRawData.eventType;
					END_IF
					IF (stEvent.stValidFields.bFromState) THEN
						stEvent.eFromState := _stNSinkRawData.fromState;
					END_IF
					IF (stEvent.stValidFields.bNotifyType) THEN
						stEvent.eNotifyType := _stNSinkRawData.notifyType;
					END_IF
					IF (stEvent.stValidFields.bToState) THEN
						stEvent.eToState := _stNSinkRawData.toState;
					END_IF
					IF (stEvent.stValidFields.bInitiatingDeviceIdentifier) THEN
						stEvent.nDeviceID := _stNSinkRawData.initiatingDeviceIdentifier;
					END_IF
					IF (stEvent.stValidFields.bNotificationClass) THEN
						stEvent.nNC := _stNSinkRawData.notificationClass;
					END_IF
					IF (stEvent.stValidFields.bPriority) THEN
						stEvent.nPriotity := _stNSinkRawData.priority;
					END_IF
					IF (stEvent.stValidFields.bProcessIdentifier) THEN
						stEvent.nProcessID := _stNSinkRawData.processIdentifier;
					END_IF
					IF (		stEvent.stValidFields.bTimeStamp
							AND	(_stNSinkRawData.timeStamp.eType = BACnetTimeStampChoice_dateTime))
					THEN
						stEvent.stDateTime := _stNSinkRawData.timeStamp.stDateTime;
					ELSE
						stEvent.stDateTime.stDate.nDay := 16#FF;
						stEvent.stDateTime.stDate.nDayOfWeek := 16#FF;
						stEvent.stDateTime.stDate.nMonth := 16#FF;
						stEvent.stDateTime.stDate.nYear := 16#FF;
						stEvent.stDateTime.stTime.nHour := 16#FF;
						stEvent.stDateTime.stTime.nMinute := 16#FF;
						stEvent.stDateTime.stTime.nSecond := 16#FF;
						stEvent.stDateTime.stTime.nHundredths := 16#FF;
					END_IF
					IF (stEvent.stValidFields.bEventObjectIdentifier) THEN
						stEvent.tObjectID := _stNSinkRawData.eventObjectIdentifier;
					END_IF
					IF (stEvent.stValidFields.bMessageText) THEN
						(* decode message text *)
						_StringExtDecode(
							pChrStringExt	:= ADR(_stNSinkRawData.messageText),
							cbOutSize		:= MIN(SIZEOF(_stNSinkRawData.messageText), SIZEOF(stEvent.sMessage)),
							pOutString		:= ADR(stEvent.sMessage),
							bValid			=> ,
							bOverflow		=> ,
							nLength			=> ,
							eSrcEncoding	=> );

						(* check overflow flag *)
						IF _StringExtDecode.bOverflow THEN
							nErrorId := BACnet_ERR_ADS_BufferSize;
	
						(* check encoding supported flag *)
						ELSIF (NOT _StringExtDecode.bValid) THEN
							nErrorId := BACnet_ERR_ADS_Encoding;
						END_IF
					END_IF

				END_IF
				(* DONE *)
				_i := 100;
			END_IF
		ELSE
			MEMSET(destAddr:=ADR(stEvent), fillByte:=0, n:=SIZEOF(stEvent));
			_fbAdsRead.bExecute := TRUE;
		END_IF

	100: (* Done *)
		bDone := (nErrorId = BACnet_ERR_NO_ERROR) AND (NOT bNoEntry);
		_i := 0;

END_CASE

(* set error flag *)
bError 	:= nErrorId > BACnet_ERR_NO_ERROR;
bBusy 	:= _i > 0;
END_FUNCTION_BLOCK

(* POU FB_BACnet_NSinkRemoveEvent, ST *)
FUNCTION_BLOCK FB_BACnet_NSinkRemoveEvent
VAR_INPUT
	bRemove		: BOOL;
	nIndex		: UDINT;
END_VAR
VAR_IN_OUT
	stAdsConn	: ST_BACnet_AdsConnection;
END_VAR
VAR_OUTPUT
	bDone		: BOOL;
	bNoEntry	: BOOL;
	bBusy		: BOOL;
	bError		: BOOL;
	nErrorId	: UINT;
END_VAR
VAR
	_fbAdsRead	: FW_AdsRead;
	_i			: INT;
	_rtrigGetSet: R_TRIG;
END_VAR
(* ADS read *)
_fbAdsRead(
	sNetId		:= stAdsConn.sAmsNetId,
	nPort		:= stAdsConn.nAmsPort,
	nIdxGrp		:= BACnet_ADSIGRP_NTFSINK_EVENTNTF_DELETE,
	nIdxOffs	:= nIndex,
	cbReadLen	:= 0,
	pReadBuff	:= 0,
	bExecute	:= ,
	tTimeout	:= BACnet_ADSTimeOut,
	bBusy		=> ,
	bError		=> ,
	nErrId		=> ,
	cbRead		=> );

(* trigger start event *)
_rtrigGetSet(CLK:= bRemove, Q=> );

(* state machine *)
CASE _i OF

	0: (* Idle *)
		IF _rtrigGetSet.Q THEN
			IF (NOT stAdsConn.bValid) THEN
				(* ADS connection not valid *)
				nErrorId := BACnet_ERR_INVALID_ADS_CONN;
			ELSIF (NOT stAdsConn.bNSink) THEN
				(* not a notification sink *)
				nErrorId := BACnet_ERR_ADS_NoNotificationSink;
			ELSE
				nErrorId := BACnet_ERR_NO_ERROR;
				_i := 1;
			END_IF
			(* reset done flag *)
			bDone := FALSE;
			(* reset no-entry flag *)
			bNoEntry := FALSE;
		END_IF
		IF (NOT bRemove) THEN
			nErrorId := BACnet_ERR_NO_ERROR;
			bDone := FALSE;
		END_IF

	(* READ *)
	1: (* read object property data over ADS *)
		IF _fbAdsRead.bExecute THEN
			IF _fbAdsRead.bError THEN
				_i := 100;
				(* entry exists? *)
				bNoEntry := ((UDINT_TO_DWORD(_fbAdsRead.nErrId) AND 16#FFF) = 16#703);
				IF (NOT bNoEntry) THEN
					nErrorId := BACnet_ERR_ADS_Read;
				END_IF
				_fbAdsRead.bExecute := FALSE;
			ELSIF (NOT _fbAdsRead.bBusy) THEN
				_fbAdsRead.bExecute := FALSE;
				(* DONE *)
				_i := 100;
			END_IF
		ELSE
			_fbAdsRead.bExecute := TRUE;
		END_IF

	100: (* Done *)
		bDone := (nErrorId = BACnet_ERR_NO_ERROR) AND (NOT bNoEntry);
		_i := 0;

END_CASE

(* set error flag *)
bError 	:= nErrorId > BACnet_ERR_NO_ERROR;
bBusy 	:= _i > 0;
END_FUNCTION_BLOCK

(* POU FB_BACnet_ObjectListProperty, ST *)
FUNCTION_BLOCK FB_BACnet_ObjectListProperty
VAR_INPUT
	bAutoGet			: BOOL:=TRUE; (* TRUE = get data from property when ADS connection OR object ID changed *)
	bGet				: BOOL; (* FALSE --> TRUE = get data from property *)
	bTypeFilter			: BOOL; (* activate input "eObjectTypeFilter" *)
	eObjType			: E_BACnetObjectType; (* select the object type that is scanned *)
END_VAR
VAR_IN_OUT
	stAdsConn			: ST_BACnet_AdsConnection;
END_VAR
VAR_OUTPUT
	bDone				: BOOL;
	bBusy				: BOOL;
	bError				: BOOL;
	nErrorId			: UINT;
	stObjIDList			: ST_BACnet_ObjectIdentifierList;
END_VAR
VAR
	_fbReadProp			: FB_BACnet_ReadProp;
	_i					: INT;
	_cbPropSize			: UDINT;
	_cbMemCpy			: UDINT;
	_nEntryCount		: UDINT;
	_iScan				: UDINT;
	_pEntry				: POINTER TO T_BACnet_ObjectIdentifier := 16#FFFFFFFF;
	_cbAdsBuf			: UDINT;
	_rtrigGetSet		: R_TRIG;
	_nAdsReloadOld		: USINT;
	_bUseObjTypeFilterOld: BOOL;
	_eObjTypeFilterOld	: E_BACnetObjectType;
	_nDeviceIdOld		: DWORD := 16#FFFFFFFF;
END_VAR
(* ADS read *);
_fbReadProp(
	BACnetDevicePort	:= stAdsConn.nAmsPort,
	bExecute			:= ,
	ObjectInstance		:= F_BACnet_GetObjInstance(stAdsConn.nDeviceId),
	ObjectType			:= BACnetObjectType_Device,
	sNetId				:= stAdsConn.sAmsNetId,
	PropertyID			:= BACnetPropertyIdentifier_ObjectList,
	DataType			:= BACnetDataType_ObjectIdentifierArr,
	ptrValue			:= ADR(stBACnet_AdsBuffer.arrData),
	nLenValue			:= SIZEOF(stBACnet_AdsBuffer.arrData),
	bDone				=> ,
	bBusy				=> ,
	bError				=> ,
	nErrID				=> ,
	nProcessedLen		=> );

(* trigger start event *)
_rtrigGetSet(CLK:= bGet, Q=> );

(* state machine *)
CASE _i OF

	0: (* Idle *)
		IF		(		(
								(_nAdsReloadOld <> stAdsConn.nReload)
							OR	(_bUseObjTypeFilterOld <> bTypeFilter)
							OR	((_eObjTypeFilterOld <> eObjType) AND bTypeFilter)
							OR	(_nDeviceIdOld <> stAdsConn.nDeviceId)
						)
					AND	bAutoGet
				)
			OR	_rtrigGetSet.Q
		THEN
			IF (NOT stAdsConn.bValid) THEN
				(* ADS connection not valid *)
				nErrorId := BACnet_ERR_INVALID_ADS_CONN;
			ELSIF (NOT stAdsConn.bServer AND NOT stAdsConn.bClient) THEN
				(* not a server nor a client *)
				nErrorId := BACnet_ERR_ADS_NoServerClient;
			ELSE
				nErrorId := BACnet_ERR_NO_ERROR;
				_i := 1;
				(* remind ADS reload counter and parameter *)
				_nAdsReloadOld := stAdsConn.nReload;
				_bUseObjTypeFilterOld := bTypeFilter;
				_eObjTypeFilterOld := eObjType;
				_nDeviceIdOld := stAdsConn.nDeviceId;
			END_IF
			(* reset done flag *)
			bDone := FALSE;
		END_IF
		IF (NOT bGet) AND (NOT bAutoGet) THEN
			nErrorId := BACnet_ERR_NO_ERROR;
			bDone := FALSE;
		END_IF

	(* READ *)
	1: (* read object property data via ADS *)
		IF TestAndSet(stBACnet_AdsBuffer.bTestSet) THEN
			IF _fbReadProp.bExecute THEN
				IF _fbReadProp.bError THEN
					_i := 100;
					nErrorId := BACnet_ERR_ADS_Read;
					_fbReadProp.bExecute := FALSE;
				ELSIF (NOT _fbReadProp.bBusy) THEN
					_fbReadProp.bExecute := FALSE;
					_cbPropSize := _fbReadProp.nProcessedLen;
					(* clear output data *)
					MEMSET(ADR(stObjIDList), 0, SIZEOF(stObjIDList));
					(* check if the ADS buffer reached its ending *)
					IF _cbPropSize > _cbAdsBuf THEN
						(* ADS buffer too small *)
						nErrorId := BACnet_ERR_ADS_BufferSize;
						(* reduce size of data to copy *)
						IF (_cbAdsBuf MOD 4) <> 0 THEN
							_cbPropSize := _F_BACnet_AlignedSize(_cbAdsBuf - 4);
						ELSE
							_cbPropSize := _cbAdsBuf;
						END_IF
					END_IF

					(* filter object type or not? *)
					IF NOT bTypeFilter THEN
						(* copy all from ADS buffer *)
						_cbMemCpy := MEMCPY(	ADR(stObjIDList.arrObjList),
												ADR(stBACnet_AdsBuffer.arrData),
												MIN(_cbPropSize, SIZEOF(stObjIDList.arrObjList))
						);
						IF _cbMemCpy < _cbPropSize THEN
							(* not all property data copied *)
							nErrorId := BACnet_ERR_ADS_TooManyObjects;
						END_IF
						(* how many entries read? *)
						stObjIDList.nEntries := _cbMemCpy / 4;
					ELSE
						(* filter - scan entry by entry *)
						_nEntryCount := _cbPropSize / 4;
						_iScan := 0;
						_pEntry := ADR(stBACnet_AdsBuffer.arrData);
						_cbPropSize := _pEntry + _cbPropSize;
						(* scan entry by entry and add to list if matching with filter *)
						WHILE (		(_pEntry + 4) <= _cbPropSize)
								AND	(_iScan < _nEntryCount)
						DO
							IF F_BACnet_GetObjType(_pEntry^) = eObjType THEN
								(* add item to list *)
								stObjIDList.arrObjList[stObjIDList.nEntries] := _pEntry^;
								stObjIDList.nEntries := stObjIDList.nEntries + 1;
							END_IF
							(* count up *)
							_iScan := _iScan + 1;
							_pEntry := _pEntry + SIZEOF(_pEntry^);
						END_WHILE
					END_IF
					(* DONE *)
					_i := 100;
				END_IF

			ELSIF (stBACnet_AdsBuffer.iLocked = 0) THEN
				_fbReadProp.bExecute := TRUE;
				(* lock global ADS buffer *)
				_cbAdsBuf := SIZEOF(stBACnet_AdsBuffer.arrData);
				stBACnet_AdsBuffer.iLocked := _cbAdsBuf;
			END_IF

			(* release temporary task lock *)
			stBACnet_AdsBuffer.bTestSet := FALSE;
		END_IF

	100: (* Done *)
		bDone := (nErrorId = BACnet_ERR_NO_ERROR);
		(* release ADS buffer *)
		stBACnet_AdsBuffer.iLocked := 0;
		_i := 0;

END_CASE

(* set error flag *)
bError 	:= nErrorId > BACnet_ERR_NO_ERROR;
bBusy 	:= _i > 0;
END_FUNCTION_BLOCK

(* POU FB_BACnet_Program, ST *)
FUNCTION_BLOCK FB_BACnet_Program
VAR_INPUT
	bRelease			: BOOL;
	bCommonError		: BOOL;
	bWaitForSomething	: BOOL;
	stDoneFlags			: ST_BACnet_ProgramHandshakeRequests;
	stFailedFlags		: ST_BACnet_ProgramHandshakeRequests;
	bModeUnloadComplex	: BOOL := TRUE;
END_VAR
VAR_IN_OUT
	Device				: FB_BACnet_Device;
END_VAR
VAR_OUTPUT
	bReady				: BOOL;
	bOverridden			: BOOL;
	bOutOfService		: BOOL;
	bFault				: BOOL;
	bInAlarm			: BOOL;
	stRequestFlags		: ST_BACnet_ProgramHandshakeRequests;
	stActiveStateFlags	: ST_BACnet_ProgramHandshakeStates;
	bError				: BOOL;
	nErrorId			: UINT;
END_VAR
VAR
(* from BACnet to PLC *)
	_ProgramChange AT%I*: WORD;			(* ~(BACnet_ProgramChange 				:		: )
											(BACnet_ObjectType 					: PROG	: ) *)
	_StatusFlags AT%I*: WORD;			(* ~(BACnet_StatusFlags 				:		: )	*)

(* from PLC to BACnet *)
	_ProgramState AT%Q*: WORD;			(* ~(BACnet_ProgramState 				:		: ) *)
	_ReasonForHalt AT%Q*: WORD;			(* ~(BACnet_ReasonForHalt 				:		: )	*)
	_SetProgramReadyState AT%Q*: BOOL;	(* ~(BACnet_SetProgramReadyState 		:		: )	*)

(* internal signals *)
	_StatusFlagsBits 	: ST_BACnet_StatusFlags;
	_bTriggerSetup		: BOOL;
	_ActiveChange		: E_BACNETPROGRAMREQUEST; (* ACTIVE PROGRAM CHANGE *)
	_bLockedForChange	: BOOL;
	_nUpdateCount		: UDINT := 0;
END_VAR
(* update server device *)
IF (Device._nUpdateCount = _nUpdateCount) THEN
	Device();
END_IF
(* remind current number of update counter *)
_nUpdateCount := Device._nUpdateCount;

(* check BitString format of StatusFlags --> if StatusFlags are less than 4, object isn't linked correctly *)
IF (_StatusFlags < 4) THEN
	(* wrong mapping *)
	nErrorId := BACnet_ERR_WRONG_MAPPING;
	bReady := FALSE;

ELSIF Device.bOperational THEN
	(* ready state *)
	bReady := TRUE;
	nErrorId := BACnet_ERR_NO_ERROR;

	(* decode status flags *)
	_StatusFlagsBits := F_BACnet_StatusFlags(_StatusFlags);

	(* copy states to output *)
	bOverridden := _StatusFlagsBits.overridden;
	bOutOfService := _StatusFlagsBits.out_of_service;
	bFault := _StatusFlagsBits.fault;
	bInAlarm := _StatusFlagsBits.in_alarm;

	(* execute change *)
	CASE _ActiveChange OF
		BACnetProgramRequest_ready:
			(* idle *);

		BACnetProgramRequest_load:
			_ProgramState	:= BACnetProgramState_loading;
			_ActiveChange	:= BACnetProgramRequest_ready;

		BACnetProgramRequest_restart,
		BACnetProgramRequest_run:
			IF _bTriggerSetup THEN
				(* wait on setup finish *)
				IF stFailedFlags.bSetup OR bCommonError OR (NOT bRelease) THEN
					(* abort *)
					_ProgramState := BACnetProgramState_halted;
					_ActiveChange := BACnetProgramRequest_ready;
					_ReasonForHalt := BACnetProgramError_progerror_internal;
				ELSIF stDoneFlags.bSetup THEN
					(* setup done, start "normal" running mode *)
					_bTriggerSetup := FALSE;
					_ActiveChange := BACnetProgramRequest_run;
				END_IF
			ELSE
				IF stFailedFlags.bRun OR bCommonError OR (NOT bRelease) THEN
					(* abort *)
					_ProgramState := BACnetProgramState_halted;
					_ActiveChange := BACnetProgramRequest_ready;
					_ReasonForHalt := BACnetProgramError_progerror_internal;
				ELSIF stDoneFlags.bRun THEN
					(* switch to running state *)
					_ProgramState := BACnetProgramState_running;
					_ActiveChange := BACnetProgramRequest_ready;
				END_IF
			END_IF

		BACnetProgramRequest_halt:
			(* wait on halted *)
			IF stFailedFlags.bHalt OR bCommonError OR (NOT bRelease) THEN
				(* abort *)
				_ProgramState := BACnetProgramState_halted;
				_ActiveChange := BACnetProgramRequest_ready;
				_ReasonForHalt := BACnetProgramError_progerror_internal;
			ELSIF stDoneFlags.bHalt THEN
				(* halted *)
				_ProgramState := BACnetProgramState_halted;
				_ActiveChange := BACnetProgramRequest_ready;
				_ReasonForHalt := BACnetProgramError_program;
			END_IF

		BACnetProgramRequest_unload:
			_ProgramState	:= BACnetProgramState_unloading;
			_ActiveChange	:= BACnetProgramRequest_ready;

	END_CASE

	(* start change request and handle error states *)
	IF (_ActiveChange = BACnetProgramRequest_ready) THEN

		CASE _ProgramState OF
			BACnetProgramState_idle:
				IF bCommonError THEN
					(* abort *)
					_ProgramState := BACnetProgramState_halted;
					_ReasonForHalt := BACnetProgramError_progerror_internal;
				ELSIF (NOT bRelease) THEN
					(* abort *)
					_ProgramState := BACnetProgramState_halted;
					_ReasonForHalt := BACnetProgramError_other;
				ELSIF (NOT _bLockedForChange) THEN
					_ReasonForHalt := BACnetProgramError_program_normal;
					CASE _ProgramChange OF
						BACnetProgramRequest_unload,
						BACnetProgramRequest_halt:
							(* acknowledge without execution *)
							_SetProgramReadyState	:= TRUE;
						BACnetProgramRequest_restart,
						BACnetProgramRequest_run,
						BACnetProgramRequest_load:
							(* execute request *)
							_ActiveChange := BACnetProgramRequest_load;
							_bTriggerSetup := TRUE;
					END_CASE
				END_IF

			BACnetProgramState_loading:
				IF bCommonError THEN
					(* abort *)
					_ProgramState := BACnetProgramState_halted;
					_ReasonForHalt := BACnetProgramError_progerror_internal;
				ELSIF (NOT bRelease) THEN
					(* abort *)
					_ProgramState := BACnetProgramState_halted;
					_ReasonForHalt := BACnetProgramError_other;
				ELSIF stFailedFlags.bLoad THEN
					(* abort *)
					_ProgramState := BACnetProgramState_halted;
					_ReasonForHalt := BACnetProgramError_load_failed;
				ELSIF stDoneFlags.bLoad THEN
					(* DONE *)
					_bTriggerSetup := TRUE;
					_ActiveChange := BACnetProgramRequest_run;
				ELSIF (NOT _bLockedForChange) THEN
					_ReasonForHalt := BACnetProgramError_program_normal;
					CASE _ProgramChange OF
						BACnetProgramRequest_load,
						BACnetProgramRequest_run,
						BACnetProgramRequest_halt,
						BACnetProgramRequest_restart:
							(* acknowledge without execution *)
							_SetProgramReadyState	:= TRUE;
						BACnetProgramRequest_unload:
							(* execute request *)
							_ActiveChange := _ProgramChange;
					END_CASE
				END_IF

			BACnetProgramState_running:
				IF bCommonError THEN
					(* abort *)
					_ProgramState := BACnetProgramState_halted;
					_ReasonForHalt := BACnetProgramError_progerror_internal;
				ELSIF (NOT bRelease) THEN
					(* abort *)
					_ProgramState := BACnetProgramState_halted;
					_ReasonForHalt := BACnetProgramError_other;
				ELSIF bWaitForSomething THEN
					(* wait on something *)
					_ProgramState := BACnetProgramState_waiting;
				ELSIF (NOT _bLockedForChange) THEN
					_ReasonForHalt := BACnetProgramError_program_normal;
					CASE _ProgramChange OF
						BACnetProgramRequest_run:
							(* is already running *)
							_SetProgramReadyState	:= TRUE;
						BACnetProgramRequest_unload,
						BACnetProgramRequest_halt:
							(* execute request *)
							_ActiveChange := _ProgramChange;
						BACnetProgramRequest_restart,
						BACnetProgramRequest_load:
							(* retrigger setup *)
							_ActiveChange := BACnetProgramRequest_restart;
							_bTriggerSetup := TRUE;
					END_CASE
				END_IF

			BACnetProgramState_waiting:
				IF bCommonError THEN
					(* abort *)
					_ProgramState := BACnetProgramState_halted;
					_ReasonForHalt := BACnetProgramError_progerror_internal;
				ELSIF (NOT bRelease) THEN
					(* abort *)
					_ProgramState := BACnetProgramState_halted;
					_ReasonForHalt := BACnetProgramError_other;
				ELSIF (NOT bWaitForSomething) THEN
					(* got it *)
					_ProgramState := BACnetProgramState_running;
				ELSIF (NOT _bLockedForChange) THEN
					_ReasonForHalt := BACnetProgramError_program_normal;
					CASE _ProgramChange OF
						BACnetProgramRequest_run:
							(* is already running *)
							_SetProgramReadyState	:= TRUE;
						BACnetProgramRequest_unload,
						BACnetProgramRequest_halt:
							(* execute request *)
							_ActiveChange := _ProgramChange;
					END_CASE
				END_IF

			BACnetProgramState_halted:
				IF (NOT bCommonError) AND bRelease AND (NOT _bLockedForChange) THEN
					CASE _ProgramChange OF
						BACnetProgramRequest_halt:
							(* acknowledge without execution *)
							_SetProgramReadyState	:= TRUE;
						BACnetProgramRequest_unload:
							(* execute request *)
							_ActiveChange := _ProgramChange;
						BACnetProgramRequest_restart,
						BACnetProgramRequest_load:
							(* retrigger setup *)
							_ActiveChange := BACnetProgramRequest_restart;
							_bTriggerSetup := TRUE;
						BACnetProgramRequest_run:
							(* start, but don't trigger setup *)
							_ActiveChange := _ProgramChange;
							_bTriggerSetup := FALSE;
					END_CASE
				END_IF

			BACnetProgramState_unloading:
				IF bModeUnloadComplex THEN
					_ReasonForHalt := BACnetProgramError_program_normal;
					IF bCommonError THEN
						(* abort *)
						_ProgramState := BACnetProgramState_halted;
						_ActiveChange := BACnetProgramRequest_ready;
						_ReasonForHalt := BACnetProgramError_progerror_internal;
					ELSIF (NOT bRelease) THEN
						(* abort *)
						_ProgramState := BACnetProgramState_halted;
						_ActiveChange := BACnetProgramRequest_ready;
						_ReasonForHalt := BACnetProgramError_other;
					ELSIF stFailedFlags.bUnload THEN
						(* abort *)
						_ProgramState := BACnetProgramState_halted;
						_ActiveChange := BACnetProgramRequest_ready;
						_ReasonForHalt := BACnetProgramError_other;
					ELSIF stDoneFlags.bUnload THEN
						(* DONE *)
						_ActiveChange := BACnetProgramRequest_ready;
						_ProgramState := BACnetProgramState_idle;
					ELSIF (NOT _bLockedForChange) THEN
						CASE _ProgramChange OF
							BACnetProgramRequest_load,
							BACnetProgramRequest_run,
							BACnetProgramRequest_halt,
							BACnetProgramRequest_restart,
							BACnetProgramRequest_unload:
								(* acknowledge without execution *)
								_SetProgramReadyState	:= TRUE;
						END_CASE
					END_IF
				END_IF

		END_CASE
	END_IF

	(* check state of "change" request *)
	IF (_ActiveChange <> BACnetProgramRequest_ready) THEN
		(* request is active, lock execution *)
		_bLockedForChange		:= TRUE;
	ELSIF _bLockedForChange AND (NOT _SetProgramReadyState) THEN
		(* change finished, tell the stack done *)
		_SetProgramReadyState	:= TRUE;
		_bTriggerSetup			:= FALSE;
	ELSIF (_ProgramChange = BACnetProgramRequest_ready) THEN
		(* wait on new requests *)
		_SetProgramReadyState	:= FALSE;
		_bLockedForChange		:= FALSE;
		_bTriggerSetup			:= FALSE;
	ELSE
		(* new request *)
		_bTriggerSetup			:= FALSE;
	END_IF

	(* external requests *)
	stRequestFlags.bLoad			:= (_ProgramState = BACnetProgramState_loading) AND (NOT _bLockedForChange);
	stRequestFlags.bSetup			:=	(		(_ActiveChange = BACnetProgramRequest_run)
										OR	(_ActiveChange = BACnetProgramRequest_restart)
									)
								AND	_bTriggerSetup;
	stRequestFlags.bRun			:= (_ActiveChange = BACnetProgramRequest_run) AND (NOT _bTriggerSetup);
	stRequestFlags.bHalt			:= _ActiveChange = BACnetProgramRequest_halt;
	stRequestFlags.bUnload		:=	(_ActiveChange = BACnetProgramRequest_unload)
								OR	(		(_ProgramState = BACnetProgramState_unloading)
										AND	(NOT _bLockedForChange)
									);

	(* active status flags *)
	stActiveStateFlags.bIdle		:= _ProgramState = BACnetProgramState_idle;
	stActiveStateFlags.bLoading		:= _ProgramState = BACnetProgramState_loading;
	stActiveStateFlags.bRunning		:= _ProgramState = BACnetProgramState_running;
	stActiveStateFlags.bWaiting		:= _ProgramState = BACnetProgramState_waiting;
	stActiveStateFlags.bHalted		:= _ProgramState = BACnetProgramState_halted;
	stActiveStateFlags.bUnloading	:= _ProgramState = BACnetProgramState_unloading;
ELSE
	(* server device not ready, reset local ready also *)
	bReady := FALSE;
	nErrorId := BACnet_ERR_OPERATIONAL;
END_IF
(* set error flag *)
bError := (nErrorId <> BACnet_ERR_NO_ERROR);
END_FUNCTION_BLOCK

(* POU FB_BACnet_Program_EX, ST *)
FUNCTION_BLOCK FB_BACnet_Program_EX
VAR_INPUT
	bRelease			: BOOL;
	bCommonError		: BOOL;
	bWaitForSomething	: BOOL;
	stDoneFlags			: ST_BACnet_ProgramHandshakeRequests;
	stFailedFlags		: ST_BACnet_ProgramHandshakeRequests;
	bModeUnloadComplex	: BOOL := TRUE;
END_VAR
VAR_IN_OUT
	Device				: FB_BACnet_Device;
END_VAR
VAR_OUTPUT
	bReady				: BOOL;
	bOverridden			: BOOL;
	bOutOfService		: BOOL;
	bFault				: BOOL;
	bInAlarm			: BOOL;
	bProcessError		: BOOL;
	bCommFailure		: BOOL;
	bOtherFault			: BOOL;
	stRequestFlags		: ST_BACnet_ProgramHandshakeRequests;
	stActiveStateFlags	: ST_BACnet_ProgramHandshakeStates;
	tObjectID			: T_BACnet_ObjectIdentifier := 16#FFFFFFFF;
	bError				: BOOL;
	nErrorId			: UINT;
END_VAR
VAR
(* from BACnet to PLC *)
	_ObjectId AT%I* : DWORD;			(* ~(BACnet_ObjectIdentifier	:		: LINK) *)
	_ProgramChange AT%I*: WORD;			(* ~(BACnet_ProgramChange 		:		: )
											(BACnet_ObjectType 			: PROG	: ) *)
	_StatusFlags AT%I*: WORD;			(* ~(BACnet_StatusFlags 		:		: )	*)
	_Reliability AT%I*: WORD;			(* ~(BACnet_Reliability 		:		: )	*)

(* from PLC to BACnet *)
	_ProgramState AT%Q*: WORD;			(* ~(BACnet_ProgramState 		:		: ) *)
	_ReasonForHalt AT%Q*: WORD;			(* ~(BACnet_ReasonForHalt 		:		: )	*)
	_SetProgramReadyState AT%Q*: BOOL;	(* ~(BACnet_SetProgramReadyState:		: )	*)

(* internal signals *)
	_StatusFlagsBits 	: ST_BACnet_StatusFlags;
	_bTriggerSetup		: BOOL;
	_ActiveChange		: E_BACNETPROGRAMREQUEST; (* ACTIVE PROGRAM CHANGE *)
	_bLockedForChange	: BOOL;
	_nUpdateCount		: UDINT := 0;
END_VAR
(* update server device *)
IF (Device._nUpdateCount = _nUpdateCount) THEN
	Device();
END_IF
(* remind current number of update counter *)
_nUpdateCount := Device._nUpdateCount;

(* check BitString format of StatusFlags --> if StatusFlags are less than 4, object isn't linked correctly *)
IF (F_BACnet_GetObjType(_ObjectId) <> BACnetObjectType_Program) THEN
	(* wrong mapping / invalid object ID *)
	IF _ObjectId = 0 THEN
		nErrorId := BACnet_ERR_WRONG_MAPPING;
	ELSE
		nErrorId := BACnet_ERR_INVALID_OBJECTID;
	END_IF
	bReady := FALSE;
	tObjectID := 16#FFFFFFFF;

ELSIF (_StatusFlags < 4) THEN
	(* wrong mapping *)
	nErrorId := BACnet_ERR_WRONG_MAPPING;
	bReady := FALSE;

ELSIF Device.bOperational THEN
	(* ready state *)
	bReady := TRUE;
	nErrorId := BACnet_ERR_NO_ERROR;

	(* decode status flags *)
	_StatusFlagsBits := F_BACnet_StatusFlags(_StatusFlags);

	(* copy states to output *)
	bOverridden := _StatusFlagsBits.overridden;
	bOutOfService := _StatusFlagsBits.out_of_service;
	bFault := _StatusFlagsBits.fault;
	bInAlarm := _StatusFlagsBits.in_alarm;
	bProcessError := (_Reliability = BACnetReliability_process_error);
	bCommFailure := (_Reliability = BACnetReliability_communication_failure);
	bOtherFault := (_Reliability = BACnetReliability_unreliable_other);
	tObjectID := _ObjectId;

	(* execute change *)
	CASE _ActiveChange OF
		BACnetProgramRequest_ready:
			(* idle *);

		BACnetProgramRequest_load:
			_ProgramState	:= BACnetProgramState_loading;
			_ActiveChange	:= BACnetProgramRequest_ready;

		BACnetProgramRequest_restart,
		BACnetProgramRequest_run:
			IF _bTriggerSetup THEN
				(* wait on setup finish *)
				IF stFailedFlags.bSetup OR bCommonError OR (NOT bRelease) THEN
					(* abort *)
					_ProgramState := BACnetProgramState_halted;
					_ActiveChange := BACnetProgramRequest_ready;
					_ReasonForHalt := BACnetProgramError_progerror_internal;
				ELSIF stDoneFlags.bSetup THEN
					(* setup done, start "normal" running mode *)
					_bTriggerSetup := FALSE;
					_ActiveChange := BACnetProgramRequest_run;
				END_IF
			ELSE
				IF stFailedFlags.bRun OR bCommonError OR (NOT bRelease) THEN
					(* abort *)
					_ProgramState := BACnetProgramState_halted;
					_ActiveChange := BACnetProgramRequest_ready;
					_ReasonForHalt := BACnetProgramError_progerror_internal;
				ELSIF stDoneFlags.bRun THEN
					(* switch to running state *)
					_ProgramState := BACnetProgramState_running;
					_ActiveChange := BACnetProgramRequest_ready;
				END_IF
			END_IF

		BACnetProgramRequest_halt:
			(* wait on halted *)
			IF stFailedFlags.bHalt OR bCommonError OR (NOT bRelease) THEN
				(* abort *)
				_ProgramState := BACnetProgramState_halted;
				_ActiveChange := BACnetProgramRequest_ready;
				_ReasonForHalt := BACnetProgramError_progerror_internal;
			ELSIF stDoneFlags.bHalt THEN
				(* halted *)
				_ProgramState := BACnetProgramState_halted;
				_ActiveChange := BACnetProgramRequest_ready;
				_ReasonForHalt := BACnetProgramError_program;
			END_IF

		BACnetProgramRequest_unload:
			_ProgramState	:= BACnetProgramState_unloading;
			_ActiveChange	:= BACnetProgramRequest_ready;

	END_CASE

	(* start change request and handle error states *)
	IF (_ActiveChange = BACnetProgramRequest_ready) THEN

		CASE _ProgramState OF
			BACnetProgramState_idle:
				IF bCommonError THEN
					(* abort *)
					_ProgramState := BACnetProgramState_halted;
					_ReasonForHalt := BACnetProgramError_progerror_internal;
				ELSIF (NOT bRelease) THEN
					(* abort *)
					_ProgramState := BACnetProgramState_halted;
					_ReasonForHalt := BACnetProgramError_other;
				ELSIF (NOT _bLockedForChange) THEN
					_ReasonForHalt := BACnetProgramError_program_normal;
					CASE _ProgramChange OF
						BACnetProgramRequest_unload,
						BACnetProgramRequest_halt:
							(* acknowledge without execution *)
							_SetProgramReadyState	:= TRUE;
						BACnetProgramRequest_restart,
						BACnetProgramRequest_run,
						BACnetProgramRequest_load:
							(* execute request *)
							_ActiveChange := BACnetProgramRequest_load;
							_bTriggerSetup := TRUE;
					END_CASE
				END_IF

			BACnetProgramState_loading:
				IF bCommonError THEN
					(* abort *)
					_ProgramState := BACnetProgramState_halted;
					_ReasonForHalt := BACnetProgramError_progerror_internal;
				ELSIF (NOT bRelease) THEN
					(* abort *)
					_ProgramState := BACnetProgramState_halted;
					_ReasonForHalt := BACnetProgramError_other;
				ELSIF stFailedFlags.bLoad THEN
					(* abort *)
					_ProgramState := BACnetProgramState_halted;
					_ReasonForHalt := BACnetProgramError_load_failed;
				ELSIF stDoneFlags.bLoad THEN
					(* DONE *)
					_bTriggerSetup := TRUE;
					_ActiveChange := BACnetProgramRequest_run;
				ELSIF (NOT _bLockedForChange) THEN
					_ReasonForHalt := BACnetProgramError_program_normal;
					CASE _ProgramChange OF
						BACnetProgramRequest_load,
						BACnetProgramRequest_run,
						BACnetProgramRequest_halt,
						BACnetProgramRequest_restart:
							(* acknowledge without execution *)
							_SetProgramReadyState	:= TRUE;
						BACnetProgramRequest_unload:
							(* execute request *)
							_ActiveChange := _ProgramChange;
					END_CASE
				END_IF

			BACnetProgramState_running:
				IF bCommonError THEN
					(* abort *)
					_ProgramState := BACnetProgramState_halted;
					_ReasonForHalt := BACnetProgramError_progerror_internal;
				ELSIF (NOT bRelease) THEN
					(* abort *)
					_ProgramState := BACnetProgramState_halted;
					_ReasonForHalt := BACnetProgramError_other;
				ELSIF bWaitForSomething THEN
					(* wait on something *)
					_ProgramState := BACnetProgramState_waiting;
				ELSIF (NOT _bLockedForChange) THEN
					_ReasonForHalt := BACnetProgramError_program_normal;
					CASE _ProgramChange OF
						BACnetProgramRequest_run:
							(* is already running *)
							_SetProgramReadyState	:= TRUE;
						BACnetProgramRequest_unload,
						BACnetProgramRequest_halt:
							(* execute request *)
							_ActiveChange := _ProgramChange;
						BACnetProgramRequest_restart,
						BACnetProgramRequest_load:
							(* retrigger setup *)
							_ActiveChange := BACnetProgramRequest_restart;
							_bTriggerSetup := TRUE;
					END_CASE
				END_IF

			BACnetProgramState_waiting:
				IF bCommonError THEN
					(* abort *)
					_ProgramState := BACnetProgramState_halted;
					_ReasonForHalt := BACnetProgramError_progerror_internal;
				ELSIF (NOT bRelease) THEN
					(* abort *)
					_ProgramState := BACnetProgramState_halted;
					_ReasonForHalt := BACnetProgramError_other;
				ELSIF (NOT bWaitForSomething) THEN
					(* got it *)
					_ProgramState := BACnetProgramState_running;
				ELSIF (NOT _bLockedForChange) THEN
					_ReasonForHalt := BACnetProgramError_program_normal;
					CASE _ProgramChange OF
						BACnetProgramRequest_run:
							(* is already running *)
							_SetProgramReadyState	:= TRUE;
						BACnetProgramRequest_unload,
						BACnetProgramRequest_halt:
							(* execute request *)
							_ActiveChange := _ProgramChange;
					END_CASE
				END_IF

			BACnetProgramState_halted:
				IF (NOT bCommonError) AND bRelease AND (NOT _bLockedForChange) THEN
					CASE _ProgramChange OF
						BACnetProgramRequest_halt:
							(* acknowledge without execution *)
							_SetProgramReadyState	:= TRUE;
						BACnetProgramRequest_unload:
							(* execute request *)
							_ActiveChange := _ProgramChange;
						BACnetProgramRequest_restart,
						BACnetProgramRequest_load:
							(* retrigger setup *)
							_ActiveChange := BACnetProgramRequest_restart;
							_bTriggerSetup := TRUE;
						BACnetProgramRequest_run:
							(* start, but don't trigger setup *)
							_ActiveChange := _ProgramChange;
							_bTriggerSetup := FALSE;
					END_CASE
				END_IF

			BACnetProgramState_unloading:
				IF bModeUnloadComplex THEN
					_ReasonForHalt := BACnetProgramError_program_normal;
					IF bCommonError THEN
						(* abort *)
						_ProgramState := BACnetProgramState_halted;
						_ActiveChange := BACnetProgramRequest_ready;
						_ReasonForHalt := BACnetProgramError_progerror_internal;
					ELSIF (NOT bRelease) THEN
						(* abort *)
						_ProgramState := BACnetProgramState_halted;
						_ActiveChange := BACnetProgramRequest_ready;
						_ReasonForHalt := BACnetProgramError_other;
					ELSIF stFailedFlags.bUnload THEN
						(* abort *)
						_ProgramState := BACnetProgramState_halted;
						_ActiveChange := BACnetProgramRequest_ready;
						_ReasonForHalt := BACnetProgramError_other;
					ELSIF stDoneFlags.bUnload THEN
						(* DONE *)
						_ActiveChange := BACnetProgramRequest_ready;
						_ProgramState := BACnetProgramState_idle;
					ELSIF (NOT _bLockedForChange) THEN
						CASE _ProgramChange OF
							BACnetProgramRequest_load,
							BACnetProgramRequest_run,
							BACnetProgramRequest_halt,
							BACnetProgramRequest_restart,
							BACnetProgramRequest_unload:
								(* acknowledge without execution *)
								_SetProgramReadyState	:= TRUE;
						END_CASE
					END_IF
				END_IF

		END_CASE
	END_IF

	(* check state of "change" request *)
	IF (_ActiveChange <> BACnetProgramRequest_ready) THEN
		(* request is active, lock execution *)
		_bLockedForChange		:= TRUE;
	ELSIF _bLockedForChange AND (NOT _SetProgramReadyState) THEN
		(* change finished, tell the stack done *)
		_SetProgramReadyState	:= TRUE;
		_bTriggerSetup			:= FALSE;
	ELSIF (_ProgramChange = BACnetProgramRequest_ready) THEN
		(* wait on new requests *)
		_SetProgramReadyState	:= FALSE;
		_bLockedForChange		:= FALSE;
		_bTriggerSetup			:= FALSE;
	ELSE
		(* new request *)
		_bTriggerSetup			:= FALSE;
	END_IF

	(* external requests *)
	stRequestFlags.bLoad			:= (_ProgramState = BACnetProgramState_loading) AND (NOT _bLockedForChange);
	stRequestFlags.bSetup			:=	(		(_ActiveChange = BACnetProgramRequest_run)
										OR	(_ActiveChange = BACnetProgramRequest_restart)
									)
								AND	_bTriggerSetup;
	stRequestFlags.bRun			:= (_ActiveChange = BACnetProgramRequest_run) AND (NOT _bTriggerSetup);
	stRequestFlags.bHalt			:= _ActiveChange = BACnetProgramRequest_halt;
	stRequestFlags.bUnload		:=	(_ActiveChange = BACnetProgramRequest_unload)
								OR	(		(_ProgramState = BACnetProgramState_unloading)
										AND	(NOT _bLockedForChange)
									);

	(* active status flags *)
	stActiveStateFlags.bIdle		:= _ProgramState = BACnetProgramState_idle;
	stActiveStateFlags.bLoading		:= _ProgramState = BACnetProgramState_loading;
	stActiveStateFlags.bRunning		:= _ProgramState = BACnetProgramState_running;
	stActiveStateFlags.bWaiting		:= _ProgramState = BACnetProgramState_waiting;
	stActiveStateFlags.bHalted		:= _ProgramState = BACnetProgramState_halted;
	stActiveStateFlags.bUnloading	:= _ProgramState = BACnetProgramState_unloading;
ELSE
	(* server device not ready, reset local ready also *)
	bReady := FALSE;
	nErrorId := BACnet_ERR_OPERATIONAL;
END_IF
(* set error flag *)
bError := (nErrorId <> BACnet_ERR_NO_ERROR);
END_FUNCTION_BLOCK

(* POU FB_BACnet_PulseConverter, ST *)
FUNCTION_BLOCK FB_BACnet_PulseConverter
VAR_IN_OUT
	Device			: FB_BACnet_Device;
END_VAR
VAR_OUTPUT
	bReady			: BOOL;
	fPresentValue	: REAL;
	nCount			: UDINT;
	bOverridden		: BOOL;
	bOutOfService	: BOOL;
	bFault			: BOOL;
	bInAlarm		: BOOL;
	bError			: BOOL;
	nErrorId		: UINT;
END_VAR
VAR
	_PresentValueIn AT%I*: REAL; 	(* ~(BACnet_PresentValue 		:		: )
								   		(BACnet_ObjectType 			: PC	: )	*)
	_Count AT%I*: UDINT;			(* ~(BACnet_Count		 		:		: ) *)
	_StatusFlags AT%I*: WORD; 		(* ~(BACnet_StatusFlags 		:		: )	*)
	_StatusFlagsBits : ST_BACnet_StatusFlags;
	_nUpdateCount : UDINT := 0;
END_VAR
(* update server device *)
IF (Device._nUpdateCount = _nUpdateCount) THEN
	Device();
END_IF
(* remind current number of update counter *)
_nUpdateCount := Device._nUpdateCount;

IF Device.bFirstCycle THEN
	(* first call of the server device since reboot/reset *)
	bReady := FALSE;

ELSIF (_StatusFlags < 4) THEN
	(* wrong mapping *)
	nErrorId := BACnet_ERR_WRONG_MAPPING;
	bReady := FALSE;

ELSIF Device.bOperational THEN
	(* ready state *)
	bReady := TRUE;
	nErrorId := BACnet_ERR_NO_ERROR;

	(* present value *)
	fPresentValue := _PresentValueIn;

	(* build bit states *)
	_StatusFlagsBits := F_BACnet_StatusFlags(_StatusFlags);

	(* copy states to output *)
	bOverridden		:= _StatusFlagsBits.overridden;
	bOutOfService	:= _StatusFlagsBits.out_of_service;
	bFault			:= _StatusFlagsBits.fault;
	bInAlarm		:= _StatusFlagsBits.in_alarm;

	(* additional information *)
	nCount			:= _Count;

ELSE
	(* server device not ready, reset local ready flag *)
	bReady := FALSE;
	nErrorId := BACnet_ERR_OPERATIONAL;
END_IF
(* set error flag *)
bError := (nErrorId <> BACnet_ERR_NO_ERROR);
END_FUNCTION_BLOCK

(* POU FB_BACnet_PulseConverter_EX, ST *)
FUNCTION_BLOCK FB_BACnet_PulseConverter_EX
VAR_IN_OUT
	Device				: FB_BACnet_Device;
END_VAR
VAR_OUTPUT
	bReady				: BOOL;
	fPresentValue		: REAL;
	bHighLimitEn		: BOOL;
	fHighLimit			: REAL;
	bLowLimitEn			: BOOL;
	fLowLimit			: REAL;
	fAdjustValue		: REAL;
	nCount				: UDINT;
	nCountBeforeChg		: UDINT;
	bOverridden			: BOOL;
	bOutOfService		: BOOL;
	bFault				: BOOL;
	bInAlarm			: BOOL;
	bOverRange			: BOOL;
	bUnderRange			: BOOL;
	bNoSensor			: BOOL;
	bOpenLoop			: BOOL;
	bShortedLoop		: BOOL;
	bCommFailure		: BOOL;
	bConfigError		: BOOL;
	bOtherFault			: BOOL;
	eEventState			: E_BACNETEVENTSTATE;
	bAckedTrans_ToOffNormal : BOOL;
	bAckedTrans_ToFault		: BOOL;
	bAckedTrans_ToNormal	: BOOL;
	tObjectID			: T_BACnet_ObjectIdentifier := 16#FFFFFFFF;
	bError				: BOOL;
	nErrorId			: UINT;
END_VAR
VAR
	_PresentValueIn AT%I*: REAL; 	(* ~(BACnet_PresentValue 		:		: )
								   		(BACnet_ObjectType 			: PC	: )	*)
	_HighLimit AT%I*: REAL;			(* ~(BACnet_HighLimit			:		: )	*)
	_LowLimit AT%I*: REAL;			(* ~(BACnet_LowLimit			:		: )	*)
	_AdjustValue AT%I*: REAL;		(* ~(BACnet_AdjustValue 		:		: ) *)
	_Count AT%I*: UDINT;			(* ~(BACnet_Count		 		:		: ) *)
	_CountBeforeChange AT%I*: UDINT;(* ~(BACnet_CountBeforeChange	:		: ) *)
	_ObjectId AT%I* : DWORD;		(* ~(BACnet_ObjectIdentifier	:		: LINK) *)
	_StatusFlags AT%I*: WORD; 		(* ~(BACnet_StatusFlags 		:		: )	*)
	_AckedTransitions AT%I*:WORD;	(* ~(BACnet_AckedTransitions	:		: ) *)
	_EventState AT%I*: WORD; 		(* ~(BACnet_EventState			:		: )	*)
	_LimitEnable AT%I*: WORD;		(* ~(BACnet_LimitEnable			:		: )	*)
	_Reliability AT%I*: WORD;		(* ~(BACnet_Reliability 		:		: )	*)
	_AckedTransBits : ST_BACnet_EventTransitionBits;
	_StatusFlagsBits : ST_BACnet_StatusFlags;
	_LimitEnableBits : ST_BACnet_LimitEnable;
	_nUpdateCount : UDINT := 0;
END_VAR
(* update server device *)
IF (Device._nUpdateCount = _nUpdateCount) THEN
	Device();
END_IF
(* remind current number of update counter *)
_nUpdateCount := Device._nUpdateCount;

IF Device.bFirstCycle THEN
	(* first call of the server device since reboot/reset *)
	bReady := FALSE;

ELSIF (F_BACnet_GetObjType(_ObjectId) <> BACnetObjectType_PulseConverter) THEN
	(* wrong mapping / invalid object ID *)
	IF _ObjectId = 0 THEN
		nErrorId := BACnet_ERR_WRONG_MAPPING;
	ELSE
		nErrorId := BACnet_ERR_INVALID_OBJECTID;
	END_IF
	bReady := FALSE;
	tObjectID := 16#FFFFFFFF;

ELSIF (_StatusFlags < 4) THEN
	(* wrong mapping *)
	nErrorId := BACnet_ERR_WRONG_MAPPING;
	bReady := FALSE;

ELSIF Device.bOperational THEN
	(* ready state *)
	bReady := TRUE;
	nErrorId := BACnet_ERR_NO_ERROR;

	(* present value *)
	fPresentValue := _PresentValueIn;

	(* build bit states *)
	_StatusFlagsBits := F_BACnet_StatusFlags(_StatusFlags);
	_AckedTransBits := F_BACnet_EventTransitionFlags(_AckedTransitions);
	_LimitEnableBits :=	F_BACnet_LimitEnableFlags(_LimitEnable);

	(* copy states to output *)
	bHighLimitEn:= _LimitEnableBits.highLimitEnable;
	bLowLimitEn	:= _LimitEnableBits.lowLimitEnable;
	bOverridden	:= _StatusFlagsBits.overridden;
	bOutOfService:= _StatusFlagsBits.out_of_service;
	bFault		:= _StatusFlagsBits.fault;
	bInAlarm	:= _StatusFlagsBits.in_alarm;
	bOverRange	:= (_Reliability = BACnetReliability_over_range);
	bUnderRange	:= (_Reliability = BACnetReliability_under_range);
	bNoSensor	:= (_Reliability = BACnetReliability_no_sensor);
	bOpenLoop	:= (_Reliability = BACnetReliability_open_loop);
	bShortedLoop:= (_Reliability = BACnetReliability_shorted_loop);
	bCommFailure := (_Reliability = BACnetReliability_communication_failure);
	bConfigError:= (_Reliability = BACnetReliability_configuration_error);
	bOtherFault	:= (_Reliability = BACnetReliability_unreliable_other);
	bAckedTrans_ToOffNormal := _AckedTransBits.to_offnormal;
	bAckedTrans_ToFault := _AckedTransBits.to_fault;
	bAckedTrans_ToNormal := _AckedTransBits.to_normal;

	(* convert enumeration *)
	eEventState := _EventState;

	(* additional information *)
	fHighLimit			:= _HighLimit;
	fLowLimit			:= _LowLimit;
	fAdjustValue		:= _AdjustValue;
	nCount				:= _Count;
	nCountBeforeChg		:= _CountBeforeChange;
	tObjectID		:= F_BACnet_GetObjInstance(_ObjectId);

ELSE
	(* server device not ready, reset local ready flag *)
	bReady := FALSE;
	nErrorId := BACnet_ERR_OPERATIONAL;
END_IF
(* set error flag *)
bError := (nErrorId <> BACnet_ERR_NO_ERROR);
END_FUNCTION_BLOCK

(* POU FB_BACnet_PulseConverter_RAW, ST *)
FUNCTION_BLOCK FB_BACnet_PulseConverter_RAW
VAR_INPUT
	nRawIn			AT%Q*: UINT; (* ~(BACnet_RawIoPulseConverterUnsignedValue : : ) *)
	bNoSensor		: BOOL;
	bOverRange		: BOOL;
	bUnderRange		: BOOL;
	bOpenLoop		: BOOL;
	bShortedLoop	: BOOL;
	bCommFailure	: BOOL;
	bConfigError	: BOOL;
	bOtherFault		: BOOL;
END_VAR
VAR_IN_OUT
	Device			: FB_BACnet_Device;
END_VAR
VAR_OUTPUT
	bReady			: BOOL;
	fPresentValue	: REAL;
	nCount			: UDINT;
	bOverridden		: BOOL;
	bOutOfService	: BOOL;
	bFault			: BOOL;
	bInAlarm		: BOOL;
	bError			: BOOL;
	nErrorId		: UINT;
END_VAR
VAR
	_PresentValueIn AT%I*: REAL; 	(* ~(BACnet_PresentValue 		:		: )
								   		(BACnet_ObjectType 			: PC	: )
										(BACnet_InputReference		: 		: nolink, disable) *)
	_Count AT%I*: UDINT;			(* ~(BACnet_Count		 		:		: ) *)
	_ObjectId AT%I*: DWORD;			(* ~(BACnet_ObjectIdentifier	:		: LINK) *)
	_StatusFlags AT%I*: WORD; 		(* ~(BACnet_StatusFlags 		:		: )	*)
	_ReliabilityIn AT%I*: WORD;		(* ~(BACnet_Reliability 		:		: )	*)
	_ReliabilityOut AT%Q*: WORD := BACnetReliability_no_fault_detected;(* ~(BACnet_Reliability 	:		: )	*)
	_StatusFlagsBits : ST_BACnet_StatusFlags;
	_nUpdateCount : UDINT := 0;
END_VAR
(* update server device *)
IF (Device._nUpdateCount = _nUpdateCount) THEN
	Device();
END_IF
(* remind current number of update counter *)
_nUpdateCount := Device._nUpdateCount;

(* handle raw error *)
IF (_ReliabilityIn <> BACnetReliability_configuration_error) THEN
	IF bNoSensor THEN
		_ReliabilityOut := BACnetReliability_no_sensor;
	ELSIF bOverRange THEN
		_ReliabilityOut := BACnetReliability_over_range;
	ELSIF bUnderRange THEN
		_ReliabilityOut := BACnetReliability_under_range;
	ELSIF bOpenLoop THEN
		_ReliabilityOut := BACnetReliability_open_loop;
	ELSIF bShortedLoop THEN
		_ReliabilityOut := BACnetReliability_shorted_loop;
	ELSIF bCommFailure THEN
		_ReliabilityOut := BACnetReliability_communication_failure;
	ELSIF bOtherFault THEN
		_ReliabilityOut := BACnetReliability_unreliable_other;
	ELSE
		_ReliabilityOut := BACnetReliability_no_fault_detected;
	END_IF
ELSE
	_ReliabilityOut := BACnetReliability_no_fault_detected;
END_IF

IF Device.bFirstCycle THEN
	(* first call of the server device since reboot/reset *)
	bReady := FALSE;

ELSIF (_StatusFlags < 4) THEN
	(* wrong mapping *)
	nErrorId := BACnet_ERR_WRONG_MAPPING;
	bReady := FALSE;

ELSIF Device.bOperational THEN
	(* ready state *)
	bReady := TRUE;
	nErrorId := BACnet_ERR_NO_ERROR;

	(* present value *)
	fPresentValue := _PresentValueIn;

	(* build bit states *)
	_StatusFlagsBits := F_BACnet_StatusFlags(_StatusFlags);

	(* copy states to output *)
	bOverridden		:= _StatusFlagsBits.overridden;
	bOutOfService	:= _StatusFlagsBits.out_of_service;
	bFault			:= _StatusFlagsBits.fault;
	bInAlarm		:= _StatusFlagsBits.in_alarm;

	(* additional information *)
	nCount			:= _Count;

ELSE
	(* server device not ready, reset local ready flag *)
	bReady := FALSE;
	nErrorId := BACnet_ERR_OPERATIONAL;
END_IF
(* set error flag *)
bError := (nErrorId <> BACnet_ERR_NO_ERROR);
END_FUNCTION_BLOCK

(* POU FB_BACnet_PWM, ST *)
FUNCTION_BLOCK FB_BACnet_PWM
VAR_INPUT
	bEnable			: BOOL;
	fPercent		: REAL; (* 0...100% *)
	tPeriod			: TIME; (* PWM period time *)
END_VAR
VAR_OUTPUT
	bEnablePV		: BOOL;
	bPresentValue	: BOOL;
END_VAR
VAR
	_fOut			: REAL;
	_tOn			: TIME;
	_tonPeriod		: TON;
	_tofOn			: TOF;
END_VAR
(* check limits *)
_fOut := LIMIT(0.0, fPercent, 100.0);

(* convert from percent value to time value in relation to period time (100% = tPara_Period, 0% = 0s) *)
_tOn := REAL_TO_TIME((_fOut / 100.0) * TIME_TO_REAL(tPeriod));

(* call period timer *)
_tonPeriod(
	IN	:= TRUE,
	PT	:= tPeriod,
	Q	=> ,
	ET	=> );

(* call on timer *)
_tofOn(
	IN	:= _tonPeriod.Q AND (_tOn > T#0ms),
	PT	:= _tOn,
	Q	=> ,
	ET	=> );

IF _tonPeriod.Q THEN
	_tonPeriod(IN:= FALSE);
	_tonPeriod(IN:= TRUE);
END_IF

(* set output *)
bPresentValue := (_tofOn.Q OR _tofOn.IN) AND bEnable;
bEnablePV := bEnable;
END_FUNCTION_BLOCK

(* POU FB_BACnet_RecipientListProperty, ST *)
FUNCTION_BLOCK FB_BACnet_RecipientListProperty
VAR_INPUT
	tObjectID			: T_BACnet_ObjectIdentifier := 16#FFFFFFFF;
	bAutoGet			: BOOL:=TRUE; (* TRUE = get data from property when ADS connection OR object ID changed *)
	bGet				: BOOL; (* FALSE --> TRUE = get data from property *)
	bSet				: BOOL; (* FALSE --> TRUE = set data into property *)
END_VAR
VAR_IN_OUT
	stAdsConn			: ST_BACnet_AdsConnection;
	stRecipients		: ST_BACnet_RecipientListDevice;
END_VAR
VAR_OUTPUT
	bDone				: BOOL;
	bBusy				: BOOL;
	bError				: BOOL;
	nErrorId			: UINT;
END_VAR
VAR
	_fbReadProp		: FB_BACnet_ReadProp;
	_fbWriteProp	: FB_BACnet_WriteProp;
	_i				: INT;
	_rtrigGet		: R_TRIG;
	_rtrigSet		: R_TRIG;

	_nAdsReloadOld	: USINT;
	_tObjectIDOld	: T_BACnet_ObjectIdentifier := 16#FFFFFFFF;

	_iEntryCheck	: UDINT;
	_iEntry			: INT;
	_iDataEntry		: INT;
	_iReadElems		: UDINT;

	_pEntryList		: POINTER TO T_BACnet_DestinationDeviceArray;

	_cbDestList		: UDINT;
	_cbDestListElem	: UDINT;
END_VAR
(*
	enum BACnetRecipient_Choice
	{
	      device,
	      address
	};
	
	typedef struct _BACnetObjectIdentifier
	{
	      union
	      {
	            struct 
	            {
	                  DWORD objInst : 22;
	                  DWORD objType : 10;
	            };
	            DWORD objId;
	      };
	}BACnetObjectIdentifier, *PBACnetObjectIdentifier;
	
	typedef struct _BACnetAddress
	{
	      BACnetAddressChoice choice;
	      BYTE layerAddress[7]; // MS/TP...LonTalk 
	      BYTE reserved;
	      USHORT      network_number;
	}BACnetAddress, *PBACnetAddress;
	
	enum BACnetAddressChoice
	{
	      Ethernet,
	      Arcnet,
	      MsTp,
	      LonTalk,
	      LonTalkNeuronId,
	      Address_3,
	      Address_4,
	      Address_5,
	      Broadcast
	};
	
	typedef struct _BACnetRecipient
	{ 
	      BACnetRecipient_Choice choiceField;
	      union
	      {
	            BACnetObjectIdentifier  device;
	            BACnetAddress           address;
	      };
	}BACnetRecipient,*PBACnetRecipient;
		
	typedef struct _BACnetDestination
	{ 
	      ULONG                              validDays;  //Bitfield of BACnetDaysOfWeek
	      BACnetTime                         fromTime;
	      BACnetTime                         toTime;
	      BACnetRecipient                    recipient;
	      ULONG                              processIdentifier;
	      DWORD                              transitionsBits;  // BACnetEventTransitionBits
	      BOOL                               issueConfirmedNotifications;
	}BACnetDestination,*PBACnetDestination;


*)

(* ADS read *)
_fbReadProp(
	BACnetDevicePort	:= stAdsConn.nAmsPort,
	bExecute			:= ,
	sNetId				:= stAdsConn.sAmsNetId,
	ObjectType			:= F_BACnet_GetObjType(tObjectID),
	PropertyID			:= BACnetPropertyIdentifier_RecipientList,
	DataType			:= BACnetDataType_RecipientArr,
	ObjectInstance		:= F_BACnet_GetObjInstance(tObjectID),
	ptrValue			:= ADR(stBACnet_AdsBuffer.arrData),
	nLenValue			:= SIZEOF(stBACnet_AdsBuffer.arrData),
	bDone				=> ,
	bBusy				=> ,
	bError				=> ,
	nErrID				=> ,
	nProcessedLen		=> );

(* ADS write *)
_fbWriteProp(
	BACnetDevicePort	:= stAdsConn.nAmsPort,
	bExecute			:= ,
	sNetId				:= stAdsConn.sAmsNetId,
	ObjectType			:= F_BACnet_GetObjType(tObjectID),
	PropertyID			:= BACnetPropertyIdentifier_RecipientList,
	Priority			:= BACnetPriority_None,
	DataType			:= BACnetDataType_RecipientArr,
	ObjectInstance		:= F_BACnet_GetObjInstance(tObjectID),
	ptrValue			:= ADR(stBACnet_AdsBuffer.arrData),
	nLenValue			:= _iDataEntry * _cbDestListElem,
	bDone				=> ,
	bBusy				=> ,
	bError				=> ,
	nErrID				=> );

(* trigger start event *)
_rtrigGet(CLK:= bGet, Q=> );
_rtrigSet(CLK:= bSet, Q=> );

(* state machine *)
CASE _i OF

	0: (* Idle *)
		IF 		_rtrigGet.Q
			OR	_rtrigSet.Q
			OR	(		(		(_nAdsReloadOld <> stAdsConn.nReload)
							OR	(_tObjectIDOld <> tObjectID)
						)
					AND	bAutoGet
				)
		THEN
			IF (NOT stAdsConn.bValid) THEN
				(* ADS connection not valid *)
				nErrorId := BACnet_ERR_INVALID_ADS_CONN;
			ELSIF (NOT stAdsConn.bServer AND NOT stAdsConn.bClient) THEN
				(* not a server nor a client *)
				nErrorId := BACnet_ERR_ADS_NoServerClient;
			ELSE
				(* decide get or set *)
				IF _rtrigGet.Q THEN
					_i := 1;
				ELSIF _rtrigSet.Q THEN
					_i := 11;
				ELSIF bAutoGet THEN
					_i := 1;
				END_IF
				nErrorId := BACnet_ERR_NO_ERROR;
				(* reset index *)
				_iEntry	:= 0;
				(* initialize pointer *)
				_pEntryList := ADR(stBACnet_AdsBuffer.arrData);
				(* remind parameter *)
				_tObjectIDOld := tObjectID;
				_nAdsReloadOld := stAdsConn.nReload;
			END_IF
			(* reset done flag *)
			bDone := FALSE;
		END_IF
		IF (NOT bGet) AND (NOT bSet) AND (NOT bAutoGet) THEN
			nErrorId := BACnet_ERR_NO_ERROR;
			bDone := FALSE;
		END_IF

	(* READ *)
	1: (* read object property data via ADS *)
		IF TestAndSet(stBACnet_AdsBuffer.bTestSet) THEN
			IF _fbReadProp.bExecute THEN
				IF _fbReadProp.bError THEN
					_i := 100;
					nErrorId := BACnet_ERR_ADS_Read;
					_fbReadProp.bExecute := FALSE;
				ELSIF (NOT _fbReadProp.bBusy) THEN
					_i := 2;
					_fbReadProp.bExecute := FALSE;
					(* clear output data *)
					MEMSET(ADR(stRecipients), 0, SIZEOF(stRecipients));
					(* check array size *)
					_cbDestList 	:= SIZEOF(_pEntryList^);
					_cbDestListElem	:= SIZEOF(_pEntryList^[0]);
					_iEntryCheck := MIN(_fbReadProp.nProcessedLen, _cbDestList) MOD _cbDestListElem;
					IF (_iEntryCheck <> 0) OR (_cbDestListElem = 0) THEN
						_i := 100;
						nErrorId := BACnet_ERR_ADS_WrongEntrySize;
					ELSE
						(* scan property *)
						_iDataEntry := 0;
						_iReadElems := MIN(32767, MIN(_fbReadProp.nProcessedLen, _cbDestList) / _cbDestListElem);
						FOR _iEntry := 0 TO UDINT_TO_INT(_iReadElems) - 1 DO
							IF		(_pEntryList^[_iEntry].stRecipient.eRecipientChoice = BACnetRecipientChoice_device)
								AND	(F_BACnet_GetObjType(_pEntryList^[_iEntry].stRecipient.tDeviceId) = BACnetObjectType_Device)
							THEN
								stRecipients.arrDestList[_iDataEntry].stFromTime	:= _pEntryList^[_iEntry].stFromTime;
								stRecipients.arrDestList[_iDataEntry].stToTime	:= _pEntryList^[_iEntry].stToTime;
								stRecipients.arrDestList[_iDataEntry].tDeviceId	:= _pEntryList^[_iEntry].stRecipient.tDeviceId;
								stRecipients.arrDestList[_iDataEntry].nProcessId	:= _pEntryList^[_iEntry].nProcessId;
								stRecipients.arrDestList[_iDataEntry].bMonday		:= _F_BACnet_IsBitFieldBitSet(_pEntryList^[_iEntry].nValidDaysFlags, BACnetDaysOfWeekBits_Monday);
								stRecipients.arrDestList[_iDataEntry].bTuesday	:= _F_BACnet_IsBitFieldBitSet(_pEntryList^[_iEntry].nValidDaysFlags, BACnetDaysOfWeekBits_Tuesday);
								stRecipients.arrDestList[_iDataEntry].bWednesday	:= _F_BACnet_IsBitFieldBitSet(_pEntryList^[_iEntry].nValidDaysFlags, BACnetDaysOfWeekBits_Wednesday);
								stRecipients.arrDestList[_iDataEntry].bThursday	:= _F_BACnet_IsBitFieldBitSet(_pEntryList^[_iEntry].nValidDaysFlags, BACnetDaysOfWeekBits_Thursday);
								stRecipients.arrDestList[_iDataEntry].bFriday		:= _F_BACnet_IsBitFieldBitSet(_pEntryList^[_iEntry].nValidDaysFlags, BACnetDaysOfWeekBits_Friday);
								stRecipients.arrDestList[_iDataEntry].bSaturday	:= _F_BACnet_IsBitFieldBitSet(_pEntryList^[_iEntry].nValidDaysFlags, BACnetDaysOfWeekBits_Saturday);
								stRecipients.arrDestList[_iDataEntry].bSunday		:= _F_BACnet_IsBitFieldBitSet(_pEntryList^[_iEntry].nValidDaysFlags, BACnetDaysOfWeekBits_Sunday);
								stRecipients.arrDestList[_iDataEntry].bToNormal	:= _F_BACnet_IsBitFieldBitSet(_pEntryList^[_iEntry].nEventTransBits, BACnetEventTransitionBit_to_normal);
								stRecipients.arrDestList[_iDataEntry].bToOffNormal:= _F_BACnet_IsBitFieldBitSet(_pEntryList^[_iEntry].nEventTransBits, BACnetEventTransitionBit_to_offnormal);
								stRecipients.arrDestList[_iDataEntry].bToFault	:= _F_BACnet_IsBitFieldBitSet(_pEntryList^[_iEntry].nEventTransBits, BACnetEventTransitionBit_to_fault);
								stRecipients.arrDestList[_iDataEntry].bIssueConfirmedNotification	:= _pEntryList^[_iEntry].bIssueConfNot;
								_iDataEntry := _iDataEntry + 1;
							END_IF
						END_FOR
						(* calculate entry count *)
						stRecipients.nEntries := _iDataEntry;
						_i := 100;
					END_IF
				END_IF

			ELSIF (stBACnet_AdsBuffer.iLocked = 0) THEN
				_fbReadProp.bExecute := TRUE;
				(* lock global ADS buffer *)
				stBACnet_AdsBuffer.iLocked := SIZEOF(stBACnet_AdsBuffer.arrData);
			END_IF

			(* release temporary task lock *)
			stBACnet_AdsBuffer.bTestSet := FALSE;
		END_IF


	(* WRITE *)
	11: (* lock global ADS buffer *)
		IF TestAndSet(stBACnet_AdsBuffer.bTestSet) THEN
			IF stBACnet_AdsBuffer.iLocked = 0 THEN
				stBACnet_AdsBuffer.iLocked := SIZEOF(stBACnet_AdsBuffer.arrData);

				(* check array size *)
				_cbDestList 	:= SIZEOF(_pEntryList^);
				_cbDestListElem	:= SIZEOF(_pEntryList^[0]);

				(* scan property *)
				_iDataEntry := 0;
				FOR _iEntry := 0 TO MIN(stRecipients.nEntries - 1, BACnet_MaxDestinationArray) DO
					IF (F_BACnet_GetObjType(stRecipients.arrDestList[_iEntry].tDeviceId) = BACnetObjectType_Device) THEN
						(* clear buffer *)
						MEMSET(ADR(_pEntryList^[_iDataEntry]), 0, _cbDestListElem);
						(* copy time and recipient information *)
						_pEntryList^[_iDataEntry].stFromTime			:= stRecipients.arrDestList[_iEntry].stFromTime;
						_pEntryList^[_iDataEntry].stToTime				:= stRecipients.arrDestList[_iEntry].stToTime;
						_pEntryList^[_iDataEntry].stRecipient.tDeviceId	:= stRecipients.arrDestList[_iEntry].tDeviceId;
						_pEntryList^[_iDataEntry].nProcessId			:= stRecipients.arrDestList[_iEntry].nProcessId;
						(* set valid days flags *)
						_pEntryList^[_iDataEntry].nValidDaysFlags := DWORD#16#00000001;
						_F_BACnet_ChangeBitFieldBit(ADR(_pEntryList^[_iDataEntry].nValidDaysFlags), BACnetDaysOfWeekBits_Monday, stRecipients.arrDestList[_iEntry].bMonday);
						_F_BACnet_ChangeBitFieldBit(ADR(_pEntryList^[_iDataEntry].nValidDaysFlags), BACnetDaysOfWeekBits_Tuesday, stRecipients.arrDestList[_iEntry].bTuesday);
						_F_BACnet_ChangeBitFieldBit(ADR(_pEntryList^[_iDataEntry].nValidDaysFlags), BACnetDaysOfWeekBits_Wednesday, stRecipients.arrDestList[_iEntry].bWednesday);
						_F_BACnet_ChangeBitFieldBit(ADR(_pEntryList^[_iDataEntry].nValidDaysFlags), BACnetDaysOfWeekBits_Thursday, stRecipients.arrDestList[_iEntry].bThursday);
						_F_BACnet_ChangeBitFieldBit(ADR(_pEntryList^[_iDataEntry].nValidDaysFlags), BACnetDaysOfWeekBits_Friday, stRecipients.arrDestList[_iEntry].bFriday);
						_F_BACnet_ChangeBitFieldBit(ADR(_pEntryList^[_iDataEntry].nValidDaysFlags), BACnetDaysOfWeekBits_Saturday, stRecipients.arrDestList[_iEntry].bSaturday);
						_F_BACnet_ChangeBitFieldBit(ADR(_pEntryList^[_iDataEntry].nValidDaysFlags), BACnetDaysOfWeekBits_Sunday, stRecipients.arrDestList[_iEntry].bSunday);
						(* set event transition flags *)
						_pEntryList^[_iDataEntry].nEventTransBits := DWORD#16#00000005;
						_F_BACnet_ChangeBitFieldBit(ADR(_pEntryList^[_iDataEntry].nEventTransBits), BACnetEventTransitionBit_to_normal, stRecipients.arrDestList[_iEntry].bToNormal);
						_F_BACnet_ChangeBitFieldBit(ADR(_pEntryList^[_iDataEntry].nEventTransBits), BACnetEventTransitionBit_to_offnormal, stRecipients.arrDestList[_iEntry].bToOffNormal);
						_F_BACnet_ChangeBitFieldBit(ADR(_pEntryList^[_iDataEntry].nEventTransBits), BACnetEventTransitionBit_to_fault, stRecipients.arrDestList[_iEntry].bToFault);
						(* set confirmed notification flag *)
						_pEntryList^[_iDataEntry].bIssueConfNot := stRecipients.arrDestList[_iEntry].bIssueConfirmedNotification;
						(* set fix choice recipient choice *)
						_pEntryList^[_iDataEntry].stRecipient.eRecipientChoice := BACnetRecipientChoice_device;
						_iDataEntry := _iDataEntry + 1;
					ELSE
						(* Wrong recipient type (device expected) *)
						nErrorId := BACnet_ERR_ADS_RecipientData;
						_i := 100;
						EXIT;
					END_IF
				END_FOR
				(* send data *)
				_i := 12;
			END_IF
			(* release temporary task lock *)
			stBACnet_AdsBuffer.bTestSet := FALSE;
		END_IF

	12:
		IF _fbWriteProp.bExecute AND (NOT _fbWriteProp.bBusy) THEN
			(* check result *)
			_fbWriteProp.bExecute := FALSE;
			IF _fbWriteProp.bError THEN
				nErrorId := BACnet_ERR_ADS_Write;
			END_IF
			_i := 100;
		ELSE
			(* start ADS write *)
			_fbWriteProp.bExecute := TRUE;
		END_IF

	100: (* Done *)
		bDone := (nErrorId = BACnet_ERR_NO_ERROR);
		(* release ADS buffer *)
		stBACnet_AdsBuffer.iLocked := 0;
		_i := 0;

END_CASE

(* set error flag *)
bError 	:= nErrorId > BACnet_ERR_NO_ERROR;
bBusy 	:= _i > 0;
END_FUNCTION_BLOCK

(* POU FB_BACnet_RemoteAccumulator, ST *)
FUNCTION_BLOCK FB_BACnet_RemoteAccumulator
VAR_IN_OUT
	RemoteDevice		: FB_BACnet_RemoteDevice;
END_VAR
VAR_OUTPUT
	bReady				: BOOL;
	nPresentValue		: UDINT;
	bOverridden			: BOOL;
	bOutOfService		: BOOL;
	bFault				: BOOL;
	bInAlarm			: BOOL;
	bError				: BOOL;
	nErrorId			: UINT;
END_VAR
VAR
	_PresentValue AT%I*:UDINT;		(* ~(BACnet_PresentValue				:		: )
										(BACnet_ObjectType					: ACC	: )
										(BACnet_RemoteCycletimeRead			: 1000	: )
										(BACnet_RemoteFlagsRead				: 1		: )
										(BACnet_RemoteResubscriptionInterval: 240	: )
                                		(BACnet_RemoteCycleTimeWrite   		: 1000	: )
                                		(BACnet_RemoteFlagsWrite       		: 1		: )	*)
	_StatusFlags AT%I*:WORD;		(* ~(BACnet_StatusFlags					:		: )	*)
	_StatusFlagsBits : ST_BACnet_StatusFlags;

	_nUpdateCount : UDINT := 0;
END_VAR
(* update client device *)
IF RemoteDevice._nUpdateCount = _nUpdateCount THEN
	RemoteDevice();
END_IF
(* remind current number of update counter *)
_nUpdateCount := RemoteDevice._nUpdateCount;

IF NOT RemoteDevice.bOperational THEN
	nErrorId := BACnet_ERR_OPERATIONAL;
	bReady := FALSE;

ELSIF _StatusFlags >= 4 THEN
	(* clear error flag *)
	nErrorId := BACnet_ERR_NO_ERROR;
	bReady := TRUE;
	(* copy present value *)
	nPresentValue := _PresentValue;

	(* build bit states *)
	_StatusFlagsBits := F_BACnet_StatusFlags(_StatusFlags);

	(* copy states to output *)
	bOverridden := _StatusFlagsBits.overridden;
	bOutOfService := _StatusFlagsBits.out_of_service;
	bFault := _StatusFlagsBits.fault;
	bInAlarm := _StatusFlagsBits.in_alarm;
ELSE
	bReady := FALSE;
	(* and set error ID *)
	nErrorId := BACnet_ERR_WRONG_MAPPING;
END_IF

(* set error flag *)
bError := (nErrorId <> BACnet_ERR_NO_ERROR);
END_FUNCTION_BLOCK

(* POU FB_BACnet_RemoteDevice, ST *)
FUNCTION_BLOCK FB_BACnet_RemoteDevice
VAR_INPUT
	bReset				: BOOL;
	bAutoReset			: BOOL;
	bDisableWOC			: BOOL;
	bReSubscribeCOV		: BOOL;
	bAutoReSubscribe	: BOOL;
	bTriggerWOC			: BOOL; (* Revision 9 feature: FALSE --> TRUE writes all output process data to remote device *)
	bReload				: BOOL; (* Reload ADS connection and increase reload counter (trigger autoget) *)
	nAmsPort			: UINT := 0; (* Optional setting: Ads port of BACnet client, default = not set *)
END_VAR
VAR_OUTPUT
	stAdsConn			: ST_BACnet_AdsConnection;
	eSystemStatus		: E_BACNETDEVICESTATUS;
	bEthLinkOk			: BOOL;
	bGatewayOk			: BOOL;
	sAmsNetId			: T_AmsNetId;
	bEnabledWOC			: BOOL;
	bWOCTriggered		: BOOL;
	bOperational		: BOOL;
	bConnecting			: BOOL;
	bFirstCycle			: BOOL;
	bError				: BOOL;
	nErrorId			: UINT;
	bClientTimeout		: BOOL;
	bServiceFailed		: BOOL;
	nTimeoutCnt			: UDINT;
	nServiceFailCnt		: UDINT;
END_VAR
VAR
	_ObjectId AT%I*:DWORD;			(* ~(BACnet_ObjectIdentifier			:		: LINK ) *)
	_SystemStatus AT%I*	: E_BACNETDEVICESTATUS;	(* ~
										(BACnet_SystemStatus 				: 		: )
										(BACnet_ObjectType					: DEV	: )
										(BACnet_RemoteCycletimeRead 		: 5000	: ) polling each 5 seconds
										(BACnet_RemoteFlagsRead        		: 2     : ) 2 = polling, so the object detects if the client is unreachable!
										(BACnet_RemoteResubscriptionInterval: 240 	: )
										(BACnet_RemoteCycleTimeWrite   		: 1000	: )
										(BACnet_RemoteFlagsWrite       		: 1		: ) *)
	_ClientStatus AT%I*:WORD;		(* ~(BACnet_ClientStatus				:		: )	*)
	_ClientControl AT%Q*:WORD;		(* ~(BACnet_ClientControl				:		: ) *)
	_rtrigReset			: R_TRIG;
	_rtrigOperational	: R_TRIG;
	_rtrigResubscribe	: R_TRIG;
	_rtrigTimeoutCnt	: R_TRIG;
	_rtrigServiceFailCnt: R_TRIG;
	_bReqResubscribe	: BOOL;
	_bComplete			: BOOL;
	_tofTimeoutLeft		: TOF;
	_tofServiceErrLeft	: TOF;
	_ftrigTimeoutLeft	: F_TRIG;

	_bHasStarted		: BOOL := TRUE;
	_nUpdateCount		: UDINT := 0;
	_nUpdateCountAdp 	: UDINT := 0;
	_BACnetAdapter		: POINTER TO FB_BACnet_Adapter;
	_AdsConn			: _FB_BACnet_AdsConn;
	_rtrigReload		: R_TRIG;
	_bLegacyMode		: BOOL;
	_tonAdsReset		: TON;

	_rtrigWOC			: R_TRIG;
	_bTriggerWOC		: BOOL;
	_tonWOCTrigger		: TON;
END_VAR
(* check pointer to bacnet adapter instance *)
IF pBACnet_Adapter > 0 THEN
	_BACnetAdapter := pBACnet_Adapter;
ELSE
	_BACnetAdapter := ADR(fbBACnet_Adapter);
END_IF

(* update server device *)
IF _BACnetAdapter^._nUpdateCount = _nUpdateCountAdp THEN
	_BACnetAdapter^();
END_IF
(* remind current number of update counter *)
_nUpdateCountAdp := _BACnetAdapter^._nUpdateCount;

(* check for client errors *)
_rtrigTimeoutCnt(CLK:= _ClientStatus.0, Q=> );
IF _rtrigTimeoutCnt.Q AND _bComplete THEN
	nErrorId := BACnet_ERR_CLIENT_TIMEOUT;
ELSIF (NOT _ClientStatus.0) THEN
	(* reset acknowledge flag *)
	_ClientControl.0 := FALSE;
END_IF
_rtrigServiceFailCnt(CLK:= _ClientStatus.1, Q=> );
IF _rtrigServiceFailCnt.Q AND _bComplete THEN
	nErrorId := BACnet_ERR_CLIENT_SERVICE;
ELSIF (NOT _ClientStatus.1) THEN
	(* reset acknowledge flag *)
	_ClientControl.1 := FALSE;
END_IF

(* convert SystemStatus to enumeration *)
eSystemStatus := _SystemStatus;
(* reset trigger *)
_rtrigReset(CLK:= bReset, Q=> );
(* reset error ID and flag *)
IF (nErrorId < 20) OR _rtrigReset.Q OR bAutoReset THEN
	nErrorId := BACnet_ERR_NO_ERROR;
END_IF
IF _rtrigReset.Q OR (NOT _bComplete) OR bAutoReset THEN
	_ClientControl.0 := _ClientStatus.0;
	_ClientControl.1 := _ClientStatus.1;
END_IF

(* read NetId and convert to string *)
sAmsNetId := _BACnetAdapter^.sAmsNetId;
(* check if it plausible *)
IF sAmsNetId = '' THEN
	(* NetId not OK, return with error *)
	nErrorId := BACnet_ERR_NO_VALID_NET_ID;
ELSIF (NOT _BACnetAdapter^.bEthLinkOk) THEN
	(* ethernet link missing *)
	nErrorId := BACnet_ERR_NO_ETH_LINK;
ELSIF (NOT _BACnetAdapter^.bGatewayOk) THEN
	(* gateway missing *)
	nErrorId := BACnet_ERR_NO_GATEWAY;
END_IF

(* summerize timeout errors *)
_tofTimeoutLeft(
	IN:= (_rtrigTimeoutCnt.Q AND _bComplete),
	PT:= T#20s,
	Q=> bClientTimeout,
	ET=> );
IF _tofTimeoutLeft.IN THEN
	nTimeoutCnt := nTimeoutCnt + 1;
END_IF
_ftrigTimeoutLeft(CLK:= _tofTimeoutLeft.Q, Q=> );

(* summerize service errors *)
_tofServiceErrLeft(
	IN:= (_rtrigServiceFailCnt.Q AND _bComplete),
	PT:= T#20s,
	Q=> bServiceFailed,
	ET=> );
IF _tofServiceErrLeft.IN THEN
	nServiceFailCnt := nServiceFailCnt + 1;
END_IF

(* WOC trigger control *)
_rtrigWOC(CLK:= bTriggerWOC, Q=> );
IF (_ClientStatus.2 OR bDisableWOC) AND bTriggerWOC THEN
	nErrorId := BACnet_ERR_WOC_DISABLED;
	_bTriggerWOC := FALSE;
ELSIF _ClientStatus.4 OR _bTriggerWOC THEN
	IF _rtrigWOC.Q THEN
		nErrorId := BACnet_ERR_WOC_TRIGGER_ACTIVE;
	ELSIF (NOT bTriggerWOC) THEN
		_bTriggerWOC := FALSE;
	END_IF
ELSIF _rtrigWOC.Q THEN
	_bTriggerWOC := TRUE;
END_IF

(* controls *)
_ClientControl.2 := bDisableWOC;
_ClientControl.3 := _bReqResubscribe;
_ClientControl.4 := _bTriggerWOC;
_ClientControl.5 := (NOT _bHasStarted); (* a-life flag *)

(* states *)
bEthLinkOk := _BACnetAdapter^.bEthLinkOk;
bGatewayOk := _BACnetAdapter^.bGatewayOk;

bEnabledWOC := (NOT _ClientStatus.2);
bConnecting := (SHR((_ClientStatus AND 16#FF00), 8) < 4);
_bComplete :=		(NOT bConnecting)
				AND	_BACnetAdapter^.bEthLinkOk;
bOperational :=		_bComplete
				AND ((NOT _ClientStatus.0) OR bAutoReset);
bWOCTriggered	:= bTriggerWOC AND _ClientStatus.4 AND (NOT (_ClientStatus.2 OR bDisableWOC));

(* Resubscribe COV *)
_rtrigOperational(CLK:= bOperational, Q=> );
_rtrigResubscribe(CLK:= bReSubscribeCOV, Q=> );
IF		(		(		(		_rtrigOperational.Q
							OR (_ftrigTimeoutLeft.Q AND bAutoReset)
						)
					AND	bAutoReSubscribe
				)
			OR	_rtrigResubscribe.Q
		)
	AND	(NOT _bReqResubscribe)
THEN
	(* operation mode reached or resubscription was externally triggered, start resubcription *)
	_bReqResubscribe	:= TRUE;
ELSIF (NOT bOperational) THEN
	(* not operational *)
	_bReqResubscribe	:= FALSE;
ELSE
	IF _bReqResubscribe AND _ClientStatus.3 THEN
		(* resubscription triggered *)
		_bReqResubscribe := FALSE;
	END_IF
END_IF

(* check WOC trigger state *)
_tonWOCTrigger(IN:= _bTriggerWOC, PT:= T#5s, Q=> , ET=> );
IF _tonWOCTrigger.Q THEN
	nErrorId := BACnet_ERR_WOC_TRIGGER_UNSUP;
	IF (NOT bTriggerWOC) THEN
		_bTriggerWOC := FALSE;
	END_IF
END_IF

(* reload ADS connection *)
_rtrigReload(CLK:= bReload, Q=> );
IF _rtrigReload.Q AND (NOT _AdsConn.bBusy) THEN
	_bLegacyMode := FALSE;
	_AdsConn(
		bAutoReload		:= FALSE,
		bReload			:= FALSE,
		bDevOperational	:= bOperational,
		sAmsNetId		:= sAmsNetId,
		tDevObjId		:= _ObjectId);
END_IF
(* probe ADS connection parameter *)
IF (NOT _bLegacyMode) AND _bComplete AND (_ObjectId <> 0) THEN
	(* call ADS connection *)
	_AdsConn(
		bAutoReload		:= TRUE,
		bReload			:=	(bReset AND (NOT _AdsConn.bReady) AND (NOT bAutoReset))
						OR	_tonAdsReset.Q
						OR	_ftrigTimeoutLeft.Q
						OR	bReload,
		bIsClient		:= TRUE,
		bDevOperational	:= bOperational,
		sAmsNetId		:= sAmsNetId,
		tDevObjId		:= _ObjectId,
		bReady			=> ,
		bBusy			=> ,
		bDone			=> ,
		bError			=> ,
		nErrorId		=> ,
		stBACnetAds		=> stAdsConn);

	(* error when ADS connection failed *)
	IF _AdsConn.bError THEN
		IF (_AdsConn.nErrorId = BACnet_ERR_ADS_LegacyStack) THEN
			_bLegacyMode := TRUE;
			stAdsConn.nReload := stAdsConn.nReload + 1;
		ELSIF (nErrorId = 0) THEN
			nErrorId := _AdsConn.nErrorId;
		END_IF
	END_IF

	(* auto reload when error is active *)
	_tonAdsReset(
		IN:=	(NOT _AdsConn.bReload)
			AND	_AdsConn.bError
			AND	bAutoReset
			AND bOperational,
		PT:= t#2s,
		Q=> ,
		ET=> );
END_IF
IF _bLegacyMode THEN
	stAdsConn.bClient	:= TRUE;
	stAdsConn.bServer	:= FALSE;
	stAdsConn.bValid	:= (nAmsPort >= 1000);
	stAdsConn.nAmsPort	:= nAmsPort;
	stAdsConn.sAmsNetId	:= sAmsNetId;
	stAdsConn.nDeviceId	:= F_BACnet_GetObjInstance(_ObjectId);
END_IF


bError := (nErrorId <> BACnet_ERR_NO_ERROR);

(* update counter *)
IF (_nUpdateCount = 0) AND _bHasStarted THEN
	bFirstCycle := TRUE;
	_bHasStarted := FALSE;
ELSE
	bFirstCycle := FALSE;
END_IF
_nUpdateCount := _nUpdateCount + 1;
END_FUNCTION_BLOCK

